DATA_BLOCK "Timer_ALARM_STOP_temp_DB"   // DB97
{ S7_Optimized_Access := 'TRUE' }
AUTHOR : Simatic
FAMILY : IEC
NAME : IEC_TMR
VERSION : 1.0
// stored: InstanceOfName IEC_TIMER
"IEC_TIMER"
BEGIN
END_DATA_BLOCK

DATA_BLOCK "Timer_PLAN_STOP_temp_DB"   // DB98
{ S7_Optimized_Access := 'TRUE' }
AUTHOR : Simatic
FAMILY : IEC
NAME : IEC_TMR
VERSION : 1.0
// stored: InstanceOfName IEC_TIMER
"IEC_TIMER"
BEGIN
END_DATA_BLOCK

DATA_BLOCK "Timer_IND_1_DB"   // DB100
{ S7_Optimized_Access := 'TRUE' }
AUTHOR : Simatic
FAMILY : IEC
NAME : IEC_TMR
VERSION : 1.0
// stored: InstanceOfName IEC_TIMER
"IEC_TIMER"
BEGIN
END_DATA_BLOCK

DATA_BLOCK "Timer_IND_2_DB"   // DB101
{ S7_Optimized_Access := 'TRUE' }
AUTHOR : Simatic
FAMILY : IEC
NAME : IEC_TMR
VERSION : 1.0
// stored: InstanceOfName IEC_TIMER
"IEC_TIMER"
BEGIN
END_DATA_BLOCK

DATA_BLOCK "TON_test_sound_DB"   // DB120
{ S7_Optimized_Access := 'TRUE' }
AUTHOR : Simatic
FAMILY : IEC
NAME : IEC_TMR
VERSION : 1.0
// stored: InstanceOfName IEC_TIMER
"IEC_TIMER"
BEGIN
END_DATA_BLOCK

DATA_BLOCK "TON_warning_1_DB"   // DB121
{ S7_Optimized_Access := 'TRUE' }
AUTHOR : Simatic
FAMILY : IEC
NAME : IEC_TMR
VERSION : 1.0
// stored: InstanceOfName IEC_TIMER
"IEC_TIMER"
BEGIN
END_DATA_BLOCK

DATA_BLOCK "TON_warning_2_DB"   // DB122
{ S7_Optimized_Access := 'TRUE' }
AUTHOR : Simatic
FAMILY : IEC
NAME : IEC_TMR
VERSION : 1.0
// stored: InstanceOfName IEC_TIMER
"IEC_TIMER"
BEGIN
END_DATA_BLOCK

DATA_BLOCK "Timer_RUN_temp_DB"   // DB124
{ S7_Optimized_Access := 'TRUE' }
AUTHOR : Simatic
FAMILY : IEC
NAME : IEC_LTMR
VERSION : 1.0
// stored: InstanceOfName IEC_LTIMER
"IEC_LTIMER"
BEGIN
END_DATA_BLOCK

// folder: (top level)

FUNCTION_BLOCK "PID_impulse"   // FB1, SCL
{ S7_Optimized_Access := 'FALSE' }
VERSION : 0.1
   VAR_INPUT
      DIR : Bool;   // Направление регулирования (1-позитивное,0-негативное)
      PV : Real;   // Величина параметра
      SP : Real;   // Величина уставки
      DB : Real;   // Зона нечувствительности
      KP : Real;   // ПИД Пропорциональный коэффициент
      TI : UDInt;   // ПИД Постоянная времени интегрирования (мс)
      TD : UDInt;   // ПИД Постоянная времени дифференцирования (мс)
      CYCLE : UDInt;   // Время цикла регулятора (мс)
      FMT : UDInt;   // Время хода исполнительного механизма (мс)
      DT_MIN : UDInt;   // Величина минимальной длительности импульса (мс)
      AUTO : Bool;   // Режим работы (0-ДИСТ, 1- АВТ)
      MORE : Bool;   // Дистанционное управление. Кнопка "Больше"
      LESS : Bool;   // Дистанционное управление. Кнопка "Меньше"
      Hold : Bool;   // (1-заморозка, 0-выполнение)
      GAP : DInt;   // Люфт
   END_VAR
   VAR_IN_OUT
      PLUS : Bool;   // Управление "Больше"
      MINUS : Bool;   // Управление "Меньше"
   END_VAR
   VAR
      BDP : Real;
      dD : Real;   // Приращение дифференциальной составляющей
      dD_max : Real;
      dI : Real;   // Приращение интегральной составляющей
      dP : Real;   // Приращение пропорциональной составляющей
      dP_1 : Real;
      dt10 : DInt;
      dt2_T : DInt;
      dt3 : DInt;
      dt3_T : DInt;
      dt4 : DInt;
      dt7 : DInt;
      dt8 : DInt;
      dt_imp_T : DInt;
      Err : Real;   // Ошибка рассогласования (t)
      Err_1 : Real;
      Err_1_T : Real;
      Ik : DInt;
      Int_reset : Bool;
      KPd : Real;
      L5 : Bool;
      L5_T : Bool;
      out : Bool;
      Pulse : Bool;   // Триггер импульса расчета
      Reset : Bool;
      TE : UDInt;   // Время цикла регулятора
      dP_T : Real;
      dI_T : Real;
      D_T : Real;
      A_N : Real := 8.0;
      A_Xf_1 : Real;
      A_Xf_2 : Real;
      D : Real;   // Приращение дифференциальной составляющей
      dD_1 : Real;
      dU : Real;   // Приращение управляющего воздействия
      dt1 : DInt;   // Длительность импульса
      dt6 : DInt;
      dt_imp : DInt;
      PLUS_T : Bool;
      MINUS_T : Bool;
      PAUSE : DInt;   // Время цикла регулятора
      L11 : Bool;
      L12 : Bool;
      Direct : Bool;   // Направление движения механизма (0-больше, 1-меньше)
   END_VAR
BEGIN
   (*Реальное время*)
   IF NOT #Reset THEN
       #TE := 0;
       #Reset := TRUE;
   ELSE
       #TE := #TE + "RT_INFO_DB".Cycle;
   END_IF;
   IF #TE >= #CYCLE AND #CYCLE <> 0 THEN
       #Pulse := TRUE;
   ELSE
       #Pulse := FALSE;
   END_IF;

   (*ПИД регулятор*)
   IF #Pulse THEN
       IF NOT #Hold THEN
           IF #AUTO THEN
               IF NOT #DIR THEN
                   #KPd := INT_TO_REAL(0) - #KP;
               ELSE
                   #KPd := #KP;
               END_IF;
               #Err := #SP - #PV;
               (*Зона нечувствительности*)
               IF ABS(#Err) < #DB / INT_TO_REAL(10) THEN
                   #Err_1 := INT_TO_REAL(0);
                   #Err_1_T := INT_TO_REAL(0);
               END_IF;
               IF ABS(#Err) > #DB / INT_TO_REAL(2) THEN
                   #Err_1 := #Err;
               END_IF;
               IF ABS(#Err) <= #DB / INT_TO_REAL(2) AND ABS(#Err) >= #DB / INT_TO_REAL(10) THEN
                   IF #Err_1_T = INT_TO_REAL(0) THEN
                       #Err_1 := INT_TO_REAL(0);
                       #Err_1_T := INT_TO_REAL(0);
                   ELSE
                       #Err_1 := #Err;
                   END_IF;
               END_IF;
               (*Д*)
               #dP := #KPd * (#Err_1 - #Err_1_T);
               (*Фильтрующий усилитель*)
               IF #TI > 0 THEN
                   #dI := #KPd * (UDINT_TO_REAL(#CYCLE) / UDINT_TO_REAL(#TI)) * ((#Err_1 + #Err_1_T) / INT_TO_REAL(2));
               ELSE
                   #dI := INT_TO_REAL(0);
               END_IF;
               (*ДД*)
               IF #TD > 0 THEN
                   (*Фильтр 1-го порядка (Апериодическое звено)*)
                   #A_Xf_1 := #A_Xf_1 + (#Err_1 - #A_Xf_1) * UDINT_TO_REAL(#CYCLE) / (UDINT_TO_REAL(#TD) / #A_N + UDINT_TO_REAL(#CYCLE));
                   (*Фильтр 2-го порядка (Апериодическое звено)*)
                   #A_Xf_2 := #A_Xf_2 + (#Err_1 - #A_Xf_1 - #A_Xf_2) * UDINT_TO_REAL(#CYCLE) / (UDINT_TO_REAL(#TD) / #A_N + UDINT_TO_REAL(#CYCLE));
                   #D := #KPd * #A_N * #A_Xf_2;
               ELSE
                   #A_Xf_1 := #Err_1;
                   #D := INT_TO_REAL(0);
               END_IF;
               #dD := #D - #D_T;
               (*Блокировка приращения пропорциональной составляющей*)
               #BDP := #KPd * #Err_1;
               IF #dP > INT_TO_REAL(0) AND #BDP < INT_TO_REAL(-100) THEN
                   #dP_1 := INT_TO_REAL(0);
               END_IF;
               IF #dP < INT_TO_REAL(0) AND #BDP > INT_TO_REAL(-100) THEN
                   #dP_1 := INT_TO_REAL(0);
               END_IF;
               IF ABS(#BDP) <= INT_TO_REAL(100) THEN
                   #dP_1 := #dP;
               END_IF;
               (*Ограничение приращений дифференциальной составляющей*)
               IF ABS(#dP_T + #dI_T) < INT_TO_REAL(100) THEN
                   #dD_max := INT_TO_REAL(100) - ABS(#dP_T + #dI_T);
               ELSE
                   #dD_max := INT_TO_REAL(0);
               END_IF;
               IF ABS(#dD) <= #dD_max THEN
                   #dD_1 := #dD;
               END_IF;
               IF #dD > #dD_max THEN
                   #dD_1 := #dD_max;
               END_IF;
               IF #dD < INT_TO_REAL(0) - #dD_max THEN
                   #dD_1 := INT_TO_REAL(0) - #dD_max;
               END_IF;
               (*Формирование ПИД закона*)
               #dU := #dP_1 + #dI + #dD_1;
               (*Ограничение амплитуды*)
               IF #dU < INT_TO_REAL(-100) THEN
                   #dU := INT_TO_REAL(-100);
               END_IF;
               IF #dU > INT_TO_REAL(100) THEN
                   #dU := INT_TO_REAL(100);
               END_IF;
               (*Расчет длительности импульса*)
               #dt1 := REAL_TO_DINT((UDINT_TO_REAL(#FMT) / INT_TO_REAL(100)) * #dU);
               (*Коррекция малых длительностей импульсов*)
               IF ABS(#dt1) < UDINT_TO_DINT(#DT_MIN) THEN
                   #dt3 := #dt1;
               ELSE
                   #dt3 := 0;
               END_IF;
               IF #dt2_T > UDINT_TO_DINT(#DT_MIN) AND ABS(#dt1) < UDINT_TO_DINT(#DT_MIN) THEN
                   #Int_reset := TRUE;
               ELSE
                   #Int_reset := FALSE;
               END_IF;
               #Ik := #Ik + #dt3;
               IF #Int_reset OR #L5_T THEN
                   #Ik := 0;
               END_IF;
               #dt4 := #dt1 + #Ik;
               IF ABS(#dt4) >= UDINT_TO_DINT(#DT_MIN) THEN
                   #L5 := TRUE;
               ELSE
                   #L5 := FALSE;
               END_IF;
               IF NOT #L5 THEN
                   #dt6 := #dt1;
               ELSE
                   #dt6 := #dt4;
               END_IF;
               (*Коррекция больших длительностей импульсов*)
               IF #dt_imp_T >= 0 THEN
                   #dt8 := UDINT_TO_DINT(#CYCLE) - #dt_imp_T;
               ELSE
                   #dt8 := - UDINT_TO_DINT(#CYCLE) - #dt_imp_T;
               END_IF;
               IF ABS(#dt8) > UDINT_TO_DINT(#CYCLE) THEN
                   #dt10 := #dt8;
               ELSE
                   #dt10 := 0;
               END_IF;
               #dt7 := #dt6 - #dt10;
               (*огр амп*)
               IF ABS(#dt7) <= UDINT_TO_DINT(#FMT) THEN
                   #dt_imp := #dt7;
               END_IF;
               IF #dt7 > UDINT_TO_DINT(#FMT) THEN
                   #dt_imp := UDINT_TO_DINT(#FMT);
               END_IF;
               IF #dt7 < - UDINT_TO_DINT(#FMT) THEN
                   #dt_imp := - UDINT_TO_DINT(#FMT);
               END_IF;
   (*Проверка ошибок*)
               ENO := TRUE;    //ENO := NOT P_ER;
           END_IF;
       ELSE
           #Err := INT_TO_REAL(0);
       END_IF;
       #Err_1_T := #Err_1;
       #dt2_T := ABS(#dt1);
       #dt3_T := #dt3;
       #dt_imp_T := #dt_imp;
       #L5_T := #L5;
       #dP_T := #dP;
       #dI_T := #dI;
       #D_T := #D;
       #TE := 0;
   END_IF;

   (* //компенсация люфта
   IF NOT #Direct AND #dt_imp < 0 THEN
       #dt_imp := #dt_imp - #GAP;
   END_IF;
   IF #Direct AND #dt_imp > 0 THEN
       #dt_imp := #dt_imp + #GAP;
   END_IF; *)

   (*Формирование ШИМ выхода*)
   IF #AUTO THEN
       IF UDINT_TO_DINT(#TE) >= ABS(#dt_imp) THEN
           #out := FALSE;
           #PLUS := false;
           #MINUS := false;
       ELSE
           #out := TRUE;
       END_IF;
       IF ABS(#dt_imp) >= UDINT_TO_DINT(#DT_MIN) THEN
           IF #dt_imp > 0 THEN
               IF #out THEN
                   #PLUS := true;
               ELSE
                   #PLUS := false;
               END_IF;
               #MINUS := false;
           ELSE
               IF #out THEN
                   #MINUS := true;
               ELSE
                   #MINUS := false;
               END_IF;
               #PLUS := false;
           END_IF;
   (*    ELSE
           #PLUS := false;
           #MINUS := false; *)
       END_IF;
   ELSE
       #PLUS := #MORE;
       #MINUS := #LESS;
   END_IF;
   (*Защита от частых коммутаций*)
   IF ((#PLUS_T AND NOT #PLUS) OR (#MINUS_T AND NOT #MINUS)) THEN
       #L11 := true;
   END_IF;
   IF #L11 THEN
       #PAUSE := UDINT_TO_DINT(#DT_MIN * INT_TO_UDINT(3));
       #L12 := true;
       #L11 := false;
   END_IF;
   IF #L12 THEN
       IF #PAUSE <= INT_TO_DINT(0) THEN
           #L12 := false;
           #PAUSE := INT_TO_DINT(0);
       ELSE
           #PAUSE := #PAUSE - UDINT_TO_DINT("RT_INFO_DB".Cycle); // / INT_TO_UDINT(10));
       END_IF;
   END_IF;
   IF #L12 AND #AUTO THEN
       #PLUS := false;
       #MINUS := false;
   END_IF;

   #PLUS_T := #PLUS;
   #MINUS_T := #MINUS;

   IF #PLUS THEN
       #Direct := FALSE;
   END_IF;
   IF #MINUS THEN
       #Direct := TRUE;
   END_IF;
END_FUNCTION_BLOCK

FUNCTION_BLOCK "PID_analog"   // FB2, SCL
{ S7_Optimized_Access := 'FALSE' }
VERSION : 0.1
   VAR_INPUT
      AUTO : Bool;   // Mode (0-manual, 1-automatic)
      DIR : Bool;   // Direction (1-positive,0-negative)
      PV : Real;   // Process variable
      SP : Real;   // Setpoint
      DB : Real;   // Deadband
      KP : Real;   // Proportional constant
      TI : UDInt;   // Integral time constant (ms)
      TD : UDInt;   // Derivative time constant (ms)
      CYCLE : UDInt;   // Cycle time (ms)
      OUT_MIN : Real;   // Output min limit (automatic mode)
      OUT_MAX : Real := 100.0;   // Output max limit (automatic mode)
      OUT_MAN : Real;   // Output (manual mode)
      Hold : Bool;   // (1-заморозка, 0-выполнение)
   END_VAR
   VAR_IN_OUT
      OUT : Real;   // Output control
   END_VAR
   VAR
      Err : Real;   // Ошибка рассогласования (t)
      Err_T : Real;   // Предыдущее значение ошибки рассогласования (t-1)
      Out_T : Real;   // Предыдущее значение выхода (t-1)
      Er : Real;   // Ошибка рассогласования (t)
      Er_T : Real;   // Предыдущее значение ошибки рассогласования (t-1)
      Integral : Real;   // Интегральная составляющая (t)
      Integral_T : Real;   // Интегральная составляющая (t-1)
      Integral_D : Real;   // Интегральное изменение
      Pulse : Bool;   // Триггер импульса расчета
      TE : UDInt;
      Reset : Bool;
      KPd : Real;
      A_N : Real := 8.0;
      A_Xf_1 : Real;
      A_Xf_2 : Real;
      Diff : Real;
   END_VAR
BEGIN
   (*Реальное время*)
   IF NOT #Reset THEN
       #TE := 0;
       #Reset := TRUE;
   ELSE
       #TE := #TE + "RT_INFO_DB".Cycle;
   END_IF;
   IF #TE >= #CYCLE AND #CYCLE <> 0 THEN
       #Pulse := TRUE;
   ELSE
       #Pulse := FALSE;
   END_IF;

   (*ПИД регулятор*)
   IF #Pulse THEN
       #Err := #SP - #PV;
       #Er := #Err;
       IF NOT #Hold THEN
           IF NOT #DIR THEN
               #KPd := INT_TO_REAL(0) - #KP;
           ELSE
               #KPd := #KP;
           END_IF;
           IF #AUTO THEN
               IF ABS(#Er) < #DB / INT_TO_REAL(10) THEN
                   #Err := INT_TO_REAL(0);
                   #Err_T := INT_TO_REAL(0);
               END_IF;
               IF ABS(#Er) > #DB / INT_TO_REAL(2) THEN
                   #Err := #Er;
               END_IF;
               IF ABS(#Er) <= #DB / INT_TO_REAL(2) AND ABS(#Er) >= #DB / INT_TO_REAL(10) THEN
                   IF #Err_T = INT_TO_REAL(0) THEN
                       #Err := INT_TO_REAL(0);
                       #Err_T := INT_TO_REAL(0);
                   ELSE
                       #Err := #Er;
                   END_IF;
               END_IF;
               IF #TI <= 0 THEN
                   #Integral_T := INT_TO_REAL(0);
                   #Integral_D := INT_TO_REAL(0);
                   #Integral := INT_TO_REAL(0);
               ELSE
                   #Integral_D := #KPd * ((#Err * UDINT_TO_REAL(#TE)) / UDINT_TO_REAL(#TI));
                   #Integral := #Integral_T + #Integral_D;
               END_IF;
               IF #TD > 0 THEN
                   (*Фильтр 1-го порядка (Апериодическое звено)*)
                   #A_Xf_1 := #A_Xf_1 + (#Err - #A_Xf_1) * UDINT_TO_REAL(#TE) / (UDINT_TO_REAL(#TD) / #A_N + UDINT_TO_REAL(#TE));
                   (*Фильтр 2-го порядка (Апериодическое звено)*)
                   #A_Xf_2 := #A_Xf_2 + (#Err - #A_Xf_1 - #A_Xf_2) * UDINT_TO_REAL(#TE) / (UDINT_TO_REAL(#TD) / #A_N + UDINT_TO_REAL(#TE));
                   #Diff := #KPd * #A_N * #A_Xf_2;
               ELSE
                   #A_Xf_1 := #Err;
                   #Diff := INT_TO_REAL(0);
               END_IF;
               #OUT := #KPd * #Err + #Integral + #Diff;
               IF #OUT < #OUT_MIN THEN
                   IF #Integral_D < INT_TO_REAL(0) THEN
                       #Integral_D := INT_TO_REAL(0);
                   END_IF;
               END_IF;
               IF #OUT > #OUT_MAX THEN
                   IF #Integral_D > INT_TO_REAL(0) THEN
                       #Integral_D := INT_TO_REAL(0);
                   END_IF;
               END_IF;
               #Integral := #Integral_T + #Integral_D;
               #OUT := #KPd * #Err + #Integral + #Diff;
               IF #OUT < #OUT_MIN THEN
                   #OUT := #OUT_MIN;
               END_IF;
               IF #OUT > #OUT_MAX THEN
                   #OUT := #OUT_MAX;
               END_IF;
           ELSE
               #OUT := #OUT_MAN;
               IF #OUT < #OUT_MIN THEN
                   #OUT := #OUT_MIN;
               END_IF;
               IF #OUT > #OUT_MAX THEN
                   #OUT := #OUT_MAX;
               END_IF;
               #Integral := #OUT - #KPd * #Err;
               #A_Xf_1 := INT_TO_REAL(0);
               #A_Xf_2 := INT_TO_REAL(0);
           END_IF;
           (*Проверка ошибок*)
           ENO := TRUE;    //ENO := NOT P_ER;
       ELSE
           #Err := INT_TO_REAL(0);
           #Err_T := INT_TO_REAL(0);
           #OUT := #OUT_MIN;
           #Integral := INT_TO_REAL(0);
       END_IF;
       #Err_T := #Err;
       #Er_T := #Er;
       #Out_T := #OUT;
       #Integral_T := #Integral;
       #TE := 0;
   END_IF;
END_FUNCTION_BLOCK

FUNCTION_BLOCK "TIME_converter"   // FB3, SCL
{ S7_Optimized_Access := 'TRUE' }
VERSION : 0.1
   VAR_INPUT
      IN : Time;   // входная переменная тип Time
   END_VAR
   VAR_OUTPUT
      Hour : Int;   // Часы
      Minute : Int;   // Минуты
      Second : Int;   // Секунды
   END_VAR
   VAR_TEMP
      in_dint_ms : DInt;
      in_dint_s : DInt;
      in_dint_m : DInt;
      in_dint_h : DInt;
   END_VAR
BEGIN
   #in_dint_ms := T_CONV(#IN);
   #in_dint_s := #in_dint_ms / 1000;
   #in_dint_m := #in_dint_s / 60;
   #in_dint_h := #in_dint_m / 60;

   #Second := DINT_TO_INT((#in_dint_s) MOD (60));
   #Minute := DINT_TO_INT((#in_dint_m) MOD (60));
   #Hour := DINT_TO_INT(#in_dint_h);
END_FUNCTION_BLOCK

FUNCTION_BLOCK "LTIME_converter"   // FB4, SCL
{ S7_Optimized_Access := 'TRUE' }
VERSION : 0.1
   VAR_INPUT
      IN : LTime;   // входная переменная тип LTime
   END_VAR
   VAR_OUTPUT
      Day : DInt;   // Дни
      Hour : Int;   // Часы
      Minute : Int;   // Минуты
      Second : Int;   // Секунды
      mSecond : Int;   // Миллисекунды
      uSecond : Int;   // Микросекунды
      nSecond : Int;   // Наносекунды
   END_VAR
   VAR_TEMP
      temp_ns : LInt;
      temp_us : LInt;
      temp_ms : LInt;
      temp_s : LInt;
      temp_m : LInt;
      temp_h : LInt;
      temp_d : LInt;
   END_VAR
BEGIN
   #temp_ns := T_CONV(#IN);
   #temp_us := #temp_ns / 1000;
   #temp_ms := #temp_us / 1000;
   #temp_s := #temp_ms / 1000;
   #temp_m := #temp_s / 60;
   #temp_h := #temp_m / 60;
   #temp_d := #temp_h / 24;

   #nSecond := LINT_TO_INT((#temp_ns) MOD (1000));
   #uSecond := LINT_TO_INT((#temp_us) MOD (1000));
   #mSecond := LINT_TO_INT((#temp_ms) MOD (1000));
   #Second := LINT_TO_INT((#temp_s) MOD (60));
   #Minute := LINT_TO_INT((#temp_m) MOD (60));
   #Hour := LINT_TO_INT((#temp_h) MOD (24));
   #Day := LINT_TO_DINT(#temp_d);
END_FUNCTION_BLOCK

FUNCTION "Read_inputs" : Void   // FC1, SCL
{ S7_Optimized_Access := 'TRUE' }
VERSION : 0.1
BEGIN
   (*ЧТЕНИЕ ВХОДОВ*)
   (*Чтение аналоговых входов*)
   (*Температура сетевой воды перед котлом*)
   IF "Sensors".T_water_before_boiler.Enable THEN
       "Read_sensor_4_20"(N_module := "Sensors".T_water_before_boiler.N_module,
                          N_chanel := "Sensors".T_water_before_boiler.N_chanel,
                          Low_limit_phisical_current := "Sensors".T_water_before_boiler.Low_limit_phisical_current,
                          High_limit_phisical_current := "Sensors".T_water_before_boiler.High_limit_phisical_current,
                          Low_limit_ADC_current := "Sensors".T_water_before_boiler.Low_limit_ADC_current,
                          High_limit_ADC_current := "Sensors".T_water_before_boiler.High_limit_ADC_current,
                          Current_ADC => "Sensors".T_water_before_boiler.Current_ADC,
                          Value => "Sensors".T_water_before_boiler.Value,
                          Alarm_sensor => "Sensors".T_water_before_boiler.Alarm_sensor,
                          Current => "Sensors".T_water_before_boiler.Current);
       //применение изменений значений точек для пересчета сигнала
       IF "Sensors".T_water_before_boiler.Apply THEN
           "Sensors".T_water_before_boiler.Low_limit_phisical_current := "Sensors".T_water_before_boiler.Low_limit_phisical_new;
           "Sensors".T_water_before_boiler.High_limit_phisical_current := "Sensors".T_water_before_boiler.High_limit_phisical_new;
           "Sensors".T_water_before_boiler.Low_limit_ADC_current := "Sensors".T_water_before_boiler.Low_limit_ADC_new;
           "Sensors".T_water_before_boiler.High_limit_ADC_current := "Sensors".T_water_before_boiler.High_limit_ADC_new;
           "Sensors".T_water_before_boiler.Apply := false;
       END_IF;
   ELSE
       "Sensors".T_water_before_boiler.Apply := false;
   END_IF;

   (*Давление сетевой воды перед котлом*)
   IF "Sensors".P_water_before_boiler.Enable THEN
       "Read_sensor_4_20"(N_module := "Sensors".P_water_before_boiler.N_module,
                          N_chanel := "Sensors".P_water_before_boiler.N_chanel,
                          Low_limit_phisical_current := "Sensors".P_water_before_boiler.Low_limit_phisical_current,
                          High_limit_phisical_current := "Sensors".P_water_before_boiler.High_limit_phisical_current,
                          Low_limit_ADC_current := "Sensors".P_water_before_boiler.Low_limit_ADC_current,
                          High_limit_ADC_current := "Sensors".P_water_before_boiler.High_limit_ADC_current,
                          Current_ADC => "Sensors".P_water_before_boiler.Current_ADC,
                          Value => "Sensors".P_water_before_boiler.Value,
                          Alarm_sensor => "Sensors".P_water_before_boiler.Alarm_sensor,
                          Current => "Sensors".P_water_before_boiler.Current);
       //применение изменений значений точек для пересчета сигнала
       IF "Sensors".P_water_before_boiler.Apply THEN
           "Sensors".P_water_before_boiler.Low_limit_phisical_current := "Sensors".P_water_before_boiler.Low_limit_phisical_new;
           "Sensors".P_water_before_boiler.High_limit_phisical_current := "Sensors".P_water_before_boiler.High_limit_phisical_new;
           "Sensors".P_water_before_boiler.Low_limit_ADC_current := "Sensors".P_water_before_boiler.Low_limit_ADC_new;
           "Sensors".P_water_before_boiler.High_limit_ADC_current := "Sensors".P_water_before_boiler.High_limit_ADC_new;
           "Sensors".P_water_before_boiler.Apply := false;
       END_IF;
   ELSE
       "Sensors".P_water_before_boiler.Apply := false;
   END_IF;

   (*Перепад давления сетевой воды через котел (кПа)*)
   IF "Sensors".dP_water_boiler.Enable THEN
       "Read_sensor_4_20"(N_module := "Sensors".dP_water_boiler.N_module,
                          N_chanel := "Sensors".dP_water_boiler.N_chanel,
                          Low_limit_phisical_current := "Sensors".dP_water_boiler.Low_limit_phisical_current,
                          High_limit_phisical_current := "Sensors".dP_water_boiler.High_limit_phisical_current,
                          Low_limit_ADC_current := "Sensors".dP_water_boiler.Low_limit_ADC_current,
                          High_limit_ADC_current := "Sensors".dP_water_boiler.High_limit_ADC_current,
                          Current_ADC => "Sensors".dP_water_boiler.Current_ADC,
                          Value => "Sensors".dP_water_boiler.Value,
                          Alarm_sensor => "Sensors".dP_water_boiler.Alarm_sensor,
                          Current => "Sensors".dP_water_boiler.Current);
       //применение изменений значений точек для пересчета сигнала
       IF "Sensors".dP_water_boiler.Apply THEN
           "Sensors".dP_water_boiler.Low_limit_phisical_current := "Sensors".dP_water_boiler.Low_limit_phisical_new;
           "Sensors".dP_water_boiler.High_limit_phisical_current := "Sensors".dP_water_boiler.High_limit_phisical_new;
           "Sensors".dP_water_boiler.Low_limit_ADC_current := "Sensors".dP_water_boiler.Low_limit_ADC_new;
           "Sensors".dP_water_boiler.High_limit_ADC_current := "Sensors".dP_water_boiler.High_limit_ADC_new;
           "Sensors".dP_water_boiler.Apply := false;
       END_IF;
   ELSE
       "Sensors".dP_water_boiler.Apply := false;
   END_IF;

   (*Температура сетевой воды после котла*)
   IF "Sensors".T_water_after_boiler.Enable THEN
       "Read_sensor_4_20"(N_module := "Sensors".T_water_after_boiler.N_module,
                          N_chanel := "Sensors".T_water_after_boiler.N_chanel,
                          Low_limit_phisical_current := "Sensors".T_water_after_boiler.Low_limit_phisical_current,
                          High_limit_phisical_current := "Sensors".T_water_after_boiler.High_limit_phisical_current,
                          Low_limit_ADC_current := "Sensors".T_water_after_boiler.Low_limit_ADC_current,
                          High_limit_ADC_current := "Sensors".T_water_after_boiler.High_limit_ADC_current,
                          Current_ADC => "Sensors".T_water_after_boiler.Current_ADC,
                          Value => "Sensors".T_water_after_boiler.Value,
                          Alarm_sensor => "Sensors".T_water_after_boiler.Alarm_sensor,
                          Current => "Sensors".T_water_after_boiler.Current);
       //применение изменений значений точек для пересчета сигнала
       IF "Sensors".T_water_after_boiler.Apply THEN
           "Sensors".T_water_after_boiler.Low_limit_phisical_current := "Sensors".T_water_after_boiler.Low_limit_phisical_new;
           "Sensors".T_water_after_boiler.High_limit_phisical_current := "Sensors".T_water_after_boiler.High_limit_phisical_new;
           "Sensors".T_water_after_boiler.Low_limit_ADC_current := "Sensors".T_water_after_boiler.Low_limit_ADC_new;
           "Sensors".T_water_after_boiler.High_limit_ADC_current := "Sensors".T_water_after_boiler.High_limit_ADC_new;
           "Sensors".T_water_after_boiler.Apply := false;
       END_IF;
   ELSE
       "Sensors".T_water_after_boiler.Apply := false;
   END_IF;

   (*Давление сетевой воды после котла*)
   IF "Sensors".P_water_after_boiler.Enable THEN
       "Read_sensor_4_20"(N_module := "Sensors".P_water_after_boiler.N_module,
                          N_chanel := "Sensors".P_water_after_boiler.N_chanel,
                          Low_limit_phisical_current := "Sensors".P_water_after_boiler.Low_limit_phisical_current,
                          High_limit_phisical_current := "Sensors".P_water_after_boiler.High_limit_phisical_current,
                          Low_limit_ADC_current := "Sensors".P_water_after_boiler.Low_limit_ADC_current,
                          High_limit_ADC_current := "Sensors".P_water_after_boiler.High_limit_ADC_current,
                          Current_ADC => "Sensors".P_water_after_boiler.Current_ADC,
                          Value => "Sensors".P_water_after_boiler.Value,
                          Alarm_sensor => "Sensors".P_water_after_boiler.Alarm_sensor,
                          Current => "Sensors".P_water_after_boiler.Current);
       //применение изменений значений точек для пересчета сигнала
       IF "Sensors".P_water_after_boiler.Apply THEN
           "Sensors".P_water_after_boiler.Low_limit_phisical_current := "Sensors".P_water_after_boiler.Low_limit_phisical_new;
           "Sensors".P_water_after_boiler.High_limit_phisical_current := "Sensors".P_water_after_boiler.High_limit_phisical_new;
           "Sensors".P_water_after_boiler.Low_limit_ADC_current := "Sensors".P_water_after_boiler.Low_limit_ADC_new;
           "Sensors".P_water_after_boiler.High_limit_ADC_current := "Sensors".P_water_after_boiler.High_limit_ADC_new;
           "Sensors".P_water_after_boiler.Apply := false;
       END_IF;
   ELSE
       "Sensors".P_water_after_boiler.Apply := false;
   END_IF;

   (*Перепад давления сетевой воды через котел (кПа)*)
   IF "Sensors".dP_water_boiler_1.Enable THEN
       "Read_sensor_4_20"(N_module := "Sensors".dP_water_boiler_1.N_module,
                          N_chanel := "Sensors".dP_water_boiler_1.N_chanel,
                          Low_limit_phisical_current := "Sensors".dP_water_boiler_1.Low_limit_phisical_current,
                          High_limit_phisical_current := "Sensors".dP_water_boiler_1.High_limit_phisical_current,
                          Low_limit_ADC_current := "Sensors".dP_water_boiler_1.Low_limit_ADC_current,
                          High_limit_ADC_current := "Sensors".dP_water_boiler_1.High_limit_ADC_current,
                          Current_ADC => "Sensors".dP_water_boiler_1.Current_ADC,
                          Value => "Sensors".dP_water_boiler_1.Value,
                          Alarm_sensor => "Sensors".dP_water_boiler_1.Alarm_sensor,
                          Current => "Sensors".dP_water_boiler_1.Current);
       //применение изменений значений точек для пересчета сигнала
       IF "Sensors".dP_water_boiler_1.Apply THEN
           "Sensors".dP_water_boiler_1.Low_limit_phisical_current := "Sensors".dP_water_boiler_1.Low_limit_phisical_new;
           "Sensors".dP_water_boiler_1.High_limit_phisical_current := "Sensors".dP_water_boiler_1.High_limit_phisical_new;
           "Sensors".dP_water_boiler_1.Low_limit_ADC_current := "Sensors".dP_water_boiler_1.Low_limit_ADC_new;
           "Sensors".dP_water_boiler_1.High_limit_ADC_current := "Sensors".dP_water_boiler_1.High_limit_ADC_new;
           "Sensors".dP_water_boiler_1.Apply := false;
       END_IF;
   ELSE
       "Sensors".dP_water_boiler_1.Apply := false;
   END_IF;

   (*Давление сетевой воды перед котлом*)
   IF "Sensors".P_water_before_boiler_1.Enable THEN
       "Read_sensor_4_20"(N_module := "Sensors".P_water_before_boiler_1.N_module,
                          N_chanel := "Sensors".P_water_before_boiler_1.N_chanel,
                          Low_limit_phisical_current := "Sensors".P_water_before_boiler_1.Low_limit_phisical_current,
                          High_limit_phisical_current := "Sensors".P_water_before_boiler_1.High_limit_phisical_current,
                          Low_limit_ADC_current := "Sensors".P_water_before_boiler_1.Low_limit_ADC_current,
                          High_limit_ADC_current := "Sensors".P_water_before_boiler_1.High_limit_ADC_current,
                          Current_ADC => "Sensors".P_water_before_boiler_1.Current_ADC,
                          Value => "Sensors".P_water_before_boiler_1.Value,
                          Alarm_sensor => "Sensors".P_water_before_boiler_1.Alarm_sensor,
                          Current => "Sensors".P_water_before_boiler_1.Current);
       //применение изменений значений точек для пересчета сигнала
       IF "Sensors".P_water_before_boiler_1.Apply THEN
           "Sensors".P_water_before_boiler_1.Low_limit_phisical_current := "Sensors".P_water_before_boiler_1.Low_limit_phisical_new;
           "Sensors".P_water_before_boiler_1.High_limit_phisical_current := "Sensors".P_water_before_boiler_1.High_limit_phisical_new;
           "Sensors".P_water_before_boiler_1.Low_limit_ADC_current := "Sensors".P_water_before_boiler_1.Low_limit_ADC_new;
           "Sensors".P_water_before_boiler_1.High_limit_ADC_current := "Sensors".P_water_before_boiler_1.High_limit_ADC_new;
           "Sensors".P_water_before_boiler_1.Apply := false;
       END_IF;
   ELSE
       "Sensors".P_water_before_boiler_1.Apply := false;
   END_IF;

   (*dP газа на котел*)
   IF "Sensors".dP_gas_boiler.Enable THEN
       "Read_sensor_4_20"(N_module := "Sensors".dP_gas_boiler.N_module,
                          N_chanel := "Sensors".dP_gas_boiler.N_chanel,
                          Low_limit_phisical_current := "Sensors".dP_gas_boiler.Low_limit_phisical_current,
                          High_limit_phisical_current := "Sensors".dP_gas_boiler.High_limit_phisical_current,
                          Low_limit_ADC_current := "Sensors".dP_gas_boiler.Low_limit_ADC_current,
                          High_limit_ADC_current := "Sensors".dP_gas_boiler.High_limit_ADC_current,
                          Current_ADC => "Sensors".dP_gas_boiler.Current_ADC,
                          Value => "Sensors".dP_gas_boiler.Value,
                          Alarm_sensor => "Sensors".dP_gas_boiler.Alarm_sensor,
                          Current => "Sensors".dP_gas_boiler.Current);
       //применение изменений значений точек для пересчета сигнала
       IF "Sensors".dP_gas_boiler.Apply THEN
           "Sensors".dP_gas_boiler.Low_limit_phisical_current := "Sensors".dP_gas_boiler.Low_limit_phisical_new;
           "Sensors".dP_gas_boiler.High_limit_phisical_current := "Sensors".dP_gas_boiler.High_limit_phisical_new;
           "Sensors".dP_gas_boiler.Low_limit_ADC_current := "Sensors".dP_gas_boiler.Low_limit_ADC_new;
           "Sensors".dP_gas_boiler.High_limit_ADC_current := "Sensors".dP_gas_boiler.High_limit_ADC_new;
           "Sensors".dP_gas_boiler.Apply := false;
       END_IF;
   ELSE
       "Sensors".dP_gas_boiler.Apply := false;
   END_IF;

   (*Разрежение в топке котла*)
   IF "Sensors".dP_furnace_boiler.Enable THEN
       "Read_sensor_4_20"(N_module := "Sensors".dP_furnace_boiler.N_module,
                          N_chanel := "Sensors".dP_furnace_boiler.N_chanel,
                          Low_limit_phisical_current := "Sensors".dP_furnace_boiler.Low_limit_phisical_current,
                          High_limit_phisical_current := "Sensors".dP_furnace_boiler.High_limit_phisical_current,
                          Low_limit_ADC_current := "Sensors".dP_furnace_boiler.Low_limit_ADC_current,
                          High_limit_ADC_current := "Sensors".dP_furnace_boiler.High_limit_ADC_current,
                          Current_ADC => "Sensors".dP_furnace_boiler.Current_ADC,
                          Value => "Sensors".dP_furnace_boiler.Value,
                          Alarm_sensor => "Sensors".dP_furnace_boiler.Alarm_sensor,
                          Current => "Sensors".dP_furnace_boiler.Current);
       //применение изменений значений точек для пересчета сигнала
       IF "Sensors".dP_furnace_boiler.Apply THEN
           "Sensors".dP_furnace_boiler.Low_limit_phisical_current := "Sensors".dP_furnace_boiler.Low_limit_phisical_new;
           "Sensors".dP_furnace_boiler.High_limit_phisical_current := "Sensors".dP_furnace_boiler.High_limit_phisical_new;
           "Sensors".dP_furnace_boiler.Low_limit_ADC_current := "Sensors".dP_furnace_boiler.Low_limit_ADC_new;
           "Sensors".dP_furnace_boiler.High_limit_ADC_current := "Sensors".dP_furnace_boiler.High_limit_ADC_new;
           "Sensors".dP_furnace_boiler.Apply := false;
       END_IF;
   ELSE
       "Sensors".dP_furnace_boiler.Apply := false;
   END_IF;

   (*Давление газа между ПЗК-1 и ПЗК-2*)
   IF "Sensors".P_gas_before_PZK1_and_PZK2.Enable THEN
       "Read_sensor_4_20"(N_module := "Sensors".P_gas_before_PZK1_and_PZK2.N_module,
                          N_chanel := "Sensors".P_gas_before_PZK1_and_PZK2.N_chanel,
                          Low_limit_phisical_current := "Sensors".P_gas_before_PZK1_and_PZK2.Low_limit_phisical_current,
                          High_limit_phisical_current := "Sensors".P_gas_before_PZK1_and_PZK2.High_limit_phisical_current,
                          Low_limit_ADC_current := "Sensors".P_gas_before_PZK1_and_PZK2.Low_limit_ADC_current,
                          High_limit_ADC_current := "Sensors".P_gas_before_PZK1_and_PZK2.High_limit_ADC_current,
                          Current_ADC => "Sensors".P_gas_before_PZK1_and_PZK2.Current_ADC,
                          Value => "Sensors".P_gas_before_PZK1_and_PZK2.Value,
                          Alarm_sensor => "Sensors".P_gas_before_PZK1_and_PZK2.Alarm_sensor,
                          Current => "Sensors".P_gas_before_PZK1_and_PZK2.Current);
       //применение изменений значений точек для пересчета сигнала
       IF "Sensors".P_gas_before_PZK1_and_PZK2.Apply THEN
           "Sensors".P_gas_before_PZK1_and_PZK2.Low_limit_phisical_current := "Sensors".P_gas_before_PZK1_and_PZK2.Low_limit_phisical_new;
           "Sensors".P_gas_before_PZK1_and_PZK2.High_limit_phisical_current := "Sensors".P_gas_before_PZK1_and_PZK2.High_limit_phisical_new;
           "Sensors".P_gas_before_PZK1_and_PZK2.Low_limit_ADC_current := "Sensors".P_gas_before_PZK1_and_PZK2.Low_limit_ADC_new;
           "Sensors".P_gas_before_PZK1_and_PZK2.High_limit_ADC_current := "Sensors".P_gas_before_PZK1_and_PZK2.High_limit_ADC_new;
           "Sensors".P_gas_before_PZK1_and_PZK2.Apply := false;
       END_IF;
   ELSE
       "Sensors".P_gas_before_PZK1_and_PZK2.Apply := false;
   END_IF;

   (*Давление газа перед горелкой*)
   IF "Sensors".P_gas_before_burner.Enable THEN
       "Read_sensor_4_20"(N_module := "Sensors".P_gas_before_burner.N_module,
                          N_chanel := "Sensors".P_gas_before_burner.N_chanel,
                          Low_limit_phisical_current := "Sensors".P_gas_before_burner.Low_limit_phisical_current,
                          High_limit_phisical_current := "Sensors".P_gas_before_burner.High_limit_phisical_current,
                          Low_limit_ADC_current := "Sensors".P_gas_before_burner.Low_limit_ADC_current,
                          High_limit_ADC_current := "Sensors".P_gas_before_burner.High_limit_ADC_current,
                          Current_ADC => "Sensors".P_gas_before_burner.Current_ADC,
                          Value => "Sensors".P_gas_before_burner.Value,
                          Alarm_sensor => "Sensors".P_gas_before_burner.Alarm_sensor,
                          Current => "Sensors".P_gas_before_burner.Current);
       //применение изменений значений точек для пересчета сигнала
       IF "Sensors".P_gas_before_burner.Apply THEN
           "Sensors".P_gas_before_burner.Low_limit_phisical_current := "Sensors".P_gas_before_burner.Low_limit_phisical_new;
           "Sensors".P_gas_before_burner.High_limit_phisical_current := "Sensors".P_gas_before_burner.High_limit_phisical_new;
           "Sensors".P_gas_before_burner.Low_limit_ADC_current := "Sensors".P_gas_before_burner.Low_limit_ADC_new;
           "Sensors".P_gas_before_burner.High_limit_ADC_current := "Sensors".P_gas_before_burner.High_limit_ADC_new;
           "Sensors".P_gas_before_burner.Apply := false;
       END_IF;
   ELSE
       "Sensors".P_gas_before_burner.Apply := false;
   END_IF;

   (*Давление воздуха к горелке*)
   IF "Sensors".P_air_burner.Enable THEN
       "Read_sensor_4_20"(N_module := "Sensors".P_air_burner.N_module,
                          N_chanel := "Sensors".P_air_burner.N_chanel,
                          Low_limit_phisical_current := "Sensors".P_air_burner.Low_limit_phisical_current,
                          High_limit_phisical_current := "Sensors".P_air_burner.High_limit_phisical_current,
                          Low_limit_ADC_current := "Sensors".P_air_burner.Low_limit_ADC_current,
                          High_limit_ADC_current := "Sensors".P_air_burner.High_limit_ADC_current,
                          Current_ADC => "Sensors".P_air_burner.Current_ADC,
                          Value => "Sensors".P_air_burner.Value,
                          Alarm_sensor => "Sensors".P_air_burner.Alarm_sensor,
                          Current => "Sensors".P_air_burner.Current);
       //применение изменений значений точек для пересчета сигнала
       IF "Sensors".P_air_burner.Apply THEN
           "Sensors".P_air_burner.Low_limit_phisical_current := "Sensors".P_air_burner.Low_limit_phisical_new;
           "Sensors".P_air_burner.High_limit_phisical_current := "Sensors".P_air_burner.High_limit_phisical_new;
           "Sensors".P_air_burner.Low_limit_ADC_current := "Sensors".P_air_burner.Low_limit_ADC_new;
           "Sensors".P_air_burner.High_limit_ADC_current := "Sensors".P_air_burner.High_limit_ADC_new;
           "Sensors".P_air_burner.Apply := false;
       END_IF;
   ELSE
       "Sensors".P_air_burner.Apply := false;
   END_IF;

   (*Температура уходящих газов*)
   IF "Sensors".T_exhaust_gas.Enable THEN
       "Read_sensor_4_20"(N_module := "Sensors".T_exhaust_gas.N_module,
                          N_chanel := "Sensors".T_exhaust_gas.N_chanel,
                          Low_limit_phisical_current := "Sensors".T_exhaust_gas.Low_limit_phisical_current,
                          High_limit_phisical_current := "Sensors".T_exhaust_gas.High_limit_phisical_current,
                          Low_limit_ADC_current := "Sensors".T_exhaust_gas.Low_limit_ADC_current,
                          High_limit_ADC_current := "Sensors".T_exhaust_gas.High_limit_ADC_current,
                          Current_ADC => "Sensors".T_exhaust_gas.Current_ADC,
                          Value => "Sensors".T_exhaust_gas.Value,
                          Alarm_sensor => "Sensors".T_exhaust_gas.Alarm_sensor,
                          Current => "Sensors".T_exhaust_gas.Current);
       //применение изменений значений точек для пересчета сигнала
       IF "Sensors".T_exhaust_gas.Apply THEN
           "Sensors".T_exhaust_gas.Low_limit_phisical_current := "Sensors".T_exhaust_gas.Low_limit_phisical_new;
           "Sensors".T_exhaust_gas.High_limit_phisical_current := "Sensors".T_exhaust_gas.High_limit_phisical_new;
           "Sensors".T_exhaust_gas.Low_limit_ADC_current := "Sensors".T_exhaust_gas.Low_limit_ADC_new;
           "Sensors".T_exhaust_gas.High_limit_ADC_current := "Sensors".T_exhaust_gas.High_limit_ADC_new;
           "Sensors".T_exhaust_gas.Apply := false;
       END_IF;
   ELSE
       "Sensors".T_exhaust_gas.Apply := false;
   END_IF;

   (*Положение рег. заслонки газа перед котлом*)
   IF "Sensors".ZRG_position.Enable THEN
       "Read_sensor_4_20"(N_module := "Sensors".ZRG_position.N_module,
                          N_chanel := "Sensors".ZRG_position.N_chanel,
                          Low_limit_phisical_current := "Sensors".ZRG_position.Low_limit_phisical_current,
                          High_limit_phisical_current := "Sensors".ZRG_position.High_limit_phisical_current,
                          Low_limit_ADC_current := "Sensors".ZRG_position.Low_limit_ADC_current,
                          High_limit_ADC_current := "Sensors".ZRG_position.High_limit_ADC_current,
                          Current_ADC => "Sensors".ZRG_position.Current_ADC,
                          Value => "Sensors".ZRG_position.Value,
                          Alarm_sensor => "Sensors".ZRG_position.Alarm_sensor,
                          Current => "Sensors".ZRG_position.Current);
       //применение изменений значений точек для пересчета сигнала
       IF "Sensors".ZRG_position.Apply THEN
           "Sensors".ZRG_position.Low_limit_phisical_current := "Sensors".ZRG_position.Low_limit_phisical_new;
           "Sensors".ZRG_position.High_limit_phisical_current := "Sensors".ZRG_position.High_limit_phisical_new;
           "Sensors".ZRG_position.Low_limit_ADC_current := "Sensors".ZRG_position.Low_limit_ADC_new;
           "Sensors".ZRG_position.High_limit_ADC_current := "Sensors".ZRG_position.High_limit_ADC_new;
           "Sensors".ZRG_position.Apply := false;
       END_IF;
   ELSE
       "Sensors".ZRG_position.Apply := false;
   END_IF;

   (*Положение направл. аппарата вентилятора*)
   IF "Sensors".NAV_position.Enable THEN
       "Read_sensor_4_20"(N_module := "Sensors".NAV_position.N_module,
                          N_chanel := "Sensors".NAV_position.N_chanel,
                          Low_limit_phisical_current := "Sensors".NAV_position.Low_limit_phisical_current,
                          High_limit_phisical_current := "Sensors".NAV_position.High_limit_phisical_current,
                          Low_limit_ADC_current := "Sensors".NAV_position.Low_limit_ADC_current,
                          High_limit_ADC_current := "Sensors".NAV_position.High_limit_ADC_current,
                          Current_ADC => "Sensors".NAV_position.Current_ADC,
                          Value => "Sensors".NAV_position.Value,
                          Alarm_sensor => "Sensors".NAV_position.Alarm_sensor,
                          Current => "Sensors".NAV_position.Current);
       //применение изменений значений точек для пересчета сигнала
       IF "Sensors".NAV_position.Apply THEN
           "Sensors".NAV_position.Low_limit_phisical_current := "Sensors".NAV_position.Low_limit_phisical_new;
           "Sensors".NAV_position.High_limit_phisical_current := "Sensors".NAV_position.High_limit_phisical_new;
           "Sensors".NAV_position.Low_limit_ADC_current := "Sensors".NAV_position.Low_limit_ADC_new;
           "Sensors".NAV_position.High_limit_ADC_current := "Sensors".NAV_position.High_limit_ADC_new;
           "Sensors".NAV_position.Apply := false;
       END_IF;
   ELSE
       "Sensors".NAV_position.Apply := false;
   END_IF;

   (*Положение направл. аппарата дымососа*)
   IF "Sensors".NAD_position.Enable THEN
       "Read_sensor_4_20"(N_module := "Sensors".NAD_position.N_module,
                          N_chanel := "Sensors".NAD_position.N_chanel,
                          Low_limit_phisical_current := "Sensors".NAD_position.Low_limit_phisical_current,
                          High_limit_phisical_current := "Sensors".NAD_position.High_limit_phisical_current,
                          Low_limit_ADC_current := "Sensors".NAD_position.Low_limit_ADC_current,
                          High_limit_ADC_current := "Sensors".NAD_position.High_limit_ADC_current,
                          Current_ADC => "Sensors".NAD_position.Current_ADC,
                          Value => "Sensors".NAD_position.Value,
                          Alarm_sensor => "Sensors".NAD_position.Alarm_sensor,
                          Current => "Sensors".NAD_position.Current);
       //применение изменений значений точек для пересчета сигнала
       IF "Sensors".NAD_position.Apply THEN
           "Sensors".NAD_position.Low_limit_phisical_current := "Sensors".NAD_position.Low_limit_phisical_new;
           "Sensors".NAD_position.High_limit_phisical_current := "Sensors".NAD_position.High_limit_phisical_new;
           "Sensors".NAD_position.Low_limit_ADC_current := "Sensors".NAD_position.Low_limit_ADC_new;
           "Sensors".NAD_position.High_limit_ADC_current := "Sensors".NAD_position.High_limit_ADC_new;
           "Sensors".NAD_position.Apply := false;
       END_IF;
   ELSE
       "Sensors".NAD_position.Apply := false;
   END_IF;

   (*Текущ. значение ПЧ ДВ*)
   IF "Sensors".DV_current_frequency.Enable THEN
       "Read_sensor_4_20"(N_module := "Sensors".DV_current_frequency.N_module,
                          N_chanel := "Sensors".DV_current_frequency.N_chanel,
                          Low_limit_phisical_current := "Sensors".DV_current_frequency.Low_limit_phisical_current,
                          High_limit_phisical_current := "Sensors".DV_current_frequency.High_limit_phisical_current,
                          Low_limit_ADC_current := "Sensors".DV_current_frequency.Low_limit_ADC_current,
                          High_limit_ADC_current := "Sensors".DV_current_frequency.High_limit_ADC_current,
                          Current_ADC => "Sensors".DV_current_frequency.Current_ADC,
                          Value => "Sensors".DV_current_frequency.Value,
                          Alarm_sensor => "Sensors".DV_current_frequency.Alarm_sensor,
                          Current => "Sensors".DV_current_frequency.Current);
       //применение изменений значений точек для пересчета сигнала
       IF "Sensors".DV_current_frequency.Apply THEN
           "Sensors".DV_current_frequency.Low_limit_phisical_current := "Sensors".DV_current_frequency.Low_limit_phisical_new;
           "Sensors".DV_current_frequency.High_limit_phisical_current := "Sensors".DV_current_frequency.High_limit_phisical_new;
           "Sensors".DV_current_frequency.Low_limit_ADC_current := "Sensors".DV_current_frequency.Low_limit_ADC_new;
           "Sensors".DV_current_frequency.High_limit_ADC_current := "Sensors".DV_current_frequency.High_limit_ADC_new;
           "Sensors".DV_current_frequency.Apply := false;
       END_IF;
   ELSE
       "Sensors".DV_current_frequency.Apply := false;
   END_IF;

   (*Текущ. значение ПЧ ДС*)
   IF "Sensors".DS_current_frequency.Enable THEN
       "Read_sensor_4_20"(N_module := "Sensors".DS_current_frequency.N_module,
                          N_chanel := "Sensors".DS_current_frequency.N_chanel,
                          Low_limit_phisical_current := "Sensors".DS_current_frequency.Low_limit_phisical_current,
                          High_limit_phisical_current := "Sensors".DS_current_frequency.High_limit_phisical_current,
                          Low_limit_ADC_current := "Sensors".DS_current_frequency.Low_limit_ADC_current,
                          High_limit_ADC_current := "Sensors".DS_current_frequency.High_limit_ADC_current,
                          Current_ADC => "Sensors".DS_current_frequency.Current_ADC,
                          Value => "Sensors".DS_current_frequency.Value,
                          Alarm_sensor => "Sensors".DS_current_frequency.Alarm_sensor,
                          Current => "Sensors".DS_current_frequency.Current);
       //применение изменений значений точек для пересчета сигнала
       IF "Sensors".DS_current_frequency.Apply THEN
           "Sensors".DS_current_frequency.Low_limit_phisical_current := "Sensors".DS_current_frequency.Low_limit_phisical_new;
           "Sensors".DS_current_frequency.High_limit_phisical_current := "Sensors".DS_current_frequency.High_limit_phisical_new;
           "Sensors".DS_current_frequency.Low_limit_ADC_current := "Sensors".DS_current_frequency.Low_limit_ADC_new;
           "Sensors".DS_current_frequency.High_limit_ADC_current := "Sensors".DS_current_frequency.High_limit_ADC_new;
           "Sensors".DS_current_frequency.Apply := false;
       END_IF;
   ELSE
       "Sensors".DS_current_frequency.Apply := false;
   END_IF;

   (*Температура газа перед БГ*)
   IF "Sensors".T_gas_before_BG.Enable THEN
       "Read_sensor_4_20"(N_module := "Sensors".T_gas_before_BG.N_module,
                          N_chanel := "Sensors".T_gas_before_BG.N_chanel,
                          Low_limit_phisical_current := "Sensors".T_gas_before_BG.Low_limit_phisical_current,
                          High_limit_phisical_current := "Sensors".T_gas_before_BG.High_limit_phisical_current,
                          Low_limit_ADC_current := "Sensors".T_gas_before_BG.Low_limit_ADC_current,
                          High_limit_ADC_current := "Sensors".T_gas_before_BG.High_limit_ADC_current,
                          Current_ADC => "Sensors".T_gas_before_BG.Current_ADC,
                          Value => "Sensors".T_gas_before_BG.Value,
                          Alarm_sensor => "Sensors".T_gas_before_BG.Alarm_sensor,
                          Current => "Sensors".T_gas_before_BG.Current);
       //применение изменений значений точек для пересчета сигнала
       IF "Sensors".T_gas_before_BG.Apply THEN
           "Sensors".T_gas_before_BG.Low_limit_phisical_current := "Sensors".T_gas_before_BG.Low_limit_phisical_new;
           "Sensors".T_gas_before_BG.High_limit_phisical_current := "Sensors".T_gas_before_BG.High_limit_phisical_new;
           "Sensors".T_gas_before_BG.Low_limit_ADC_current := "Sensors".T_gas_before_BG.Low_limit_ADC_new;
           "Sensors".T_gas_before_BG.High_limit_ADC_current := "Sensors".T_gas_before_BG.High_limit_ADC_new;
           "Sensors".T_gas_before_BG.Apply := false;
       END_IF;
   ELSE
       "Sensors".T_gas_before_BG.Apply := false;
   END_IF;

   (*Давление газа перед БГ*)
   IF "Sensors".P_gas_before_BG.Enable THEN
       "Read_sensor_4_20"(N_module := "Sensors".P_gas_before_BG.N_module,
                          N_chanel := "Sensors".P_gas_before_BG.N_chanel,
                          Low_limit_phisical_current := "Sensors".P_gas_before_BG.Low_limit_phisical_current,
                          High_limit_phisical_current := "Sensors".P_gas_before_BG.High_limit_phisical_current,
                          Low_limit_ADC_current := "Sensors".P_gas_before_BG.Low_limit_ADC_current,
                          High_limit_ADC_current := "Sensors".P_gas_before_BG.High_limit_ADC_current,
                          Current_ADC => "Sensors".P_gas_before_BG.Current_ADC,
                          Value => "Sensors".P_gas_before_BG.Value,
                          Alarm_sensor => "Sensors".P_gas_before_BG.Alarm_sensor,
                          Current => "Sensors".P_gas_before_BG.Current);
       //применение изменений значений точек для пересчета сигнала
       IF "Sensors".P_gas_before_BG.Apply THEN
           "Sensors".P_gas_before_BG.Low_limit_phisical_current := "Sensors".P_gas_before_BG.Low_limit_phisical_new;
           "Sensors".P_gas_before_BG.High_limit_phisical_current := "Sensors".P_gas_before_BG.High_limit_phisical_new;
           "Sensors".P_gas_before_BG.Low_limit_ADC_current := "Sensors".P_gas_before_BG.Low_limit_ADC_new;
           "Sensors".P_gas_before_BG.High_limit_ADC_current := "Sensors".P_gas_before_BG.High_limit_ADC_new;
           "Sensors".P_gas_before_BG.Apply := false;
       END_IF;
   ELSE
       "Sensors".P_gas_before_BG.Apply := false;
   END_IF;


   (*Чтение дискретных входов*)
   (*Наличие пламени горелки*)
   IF "Sensors".Burner_flame.Enable THEN
       "Read_discret_signal"(N_module := "Sensors".Burner_flame.N_module,
                             N_chanel := "Sensors".Burner_flame.N_chanel,
                             Invert := "Sensors".Burner_flame.Invert,
                             Value => "Sensors".Burner_flame.Value);
   ELSE
       "Sensors".Burner_flame.Value := false;
   END_IF;

   (*Наличие пламени запальника горелки*)
   IF "Sensors".Igniter_flame.Enable THEN
       "Read_discret_signal"(N_module := "Sensors".Igniter_flame.N_module,
                             N_chanel := "Sensors".Igniter_flame.N_chanel,
                             Invert := "Sensors".Igniter_flame.Invert,
                             Value => "Sensors".Igniter_flame.Value);
   ELSE
       "Sensors".Igniter_flame.Value := false;
   END_IF;

   (*Клапан безопасности закрыт*)
   IF "Sensors".KB_close.Enable THEN
       "Read_discret_signal"(N_module := "Sensors".KB_close.N_module,
                             N_chanel := "Sensors".KB_close.N_chanel,
                             Invert := "Sensors".KB_close.Invert,
                             Value => "Sensors".KB_close.Value);
   ELSE
       "Sensors".KB_close.Value := false;
   END_IF;

   (*Клапан опрессовки открыт*)
   IF "Sensors".KO_open.Enable THEN
       "Read_discret_signal"(N_module := "Sensors".KO_open.N_module,
                             N_chanel := "Sensors".KO_open.N_chanel,
                             Invert := "Sensors".KO_open.Invert,
                             Value => "Sensors".KO_open.Value);
   ELSE
       "Sensors".KO_open.Value := false;
   END_IF;

   (*Клапан запальника открыт*)
   IF "Sensors".KZ_open.Enable THEN
       "Read_discret_signal"(N_module := "Sensors".KZ_open.N_module,
                             N_chanel := "Sensors".KZ_open.N_chanel,
                             Invert := "Sensors".KZ_open.Invert,
                             Value => "Sensors".KZ_open.Value);
   ELSE
       "Sensors".KZ_open.Value := false;
   END_IF;

   (*ПЗК-1 горелки открыт*)
   IF "Sensors".PZK1_open.Enable THEN
       "Read_discret_signal"(N_module := "Sensors".PZK1_open.N_module,
                             N_chanel := "Sensors".PZK1_open.N_chanel,
                             Invert := "Sensors".PZK1_open.Invert,
                             Value => "Sensors".PZK1_open.Value);
   ELSE
       "Sensors".PZK1_open.Value := false;
   END_IF;

   (*ПЗК-2 горелки не закрыт*)
   IF "Sensors".PZK2_not_close.Enable THEN
       "Read_discret_signal"(N_module := "Sensors".PZK2_not_close.N_module,
                             N_chanel := "Sensors".PZK2_not_close.N_chanel,
                             Invert := "Sensors".PZK2_not_close.Invert,
                             Value => "Sensors".PZK2_not_close.Value);
   ELSE
       "Sensors".PZK2_not_close.Value := false;
   END_IF;

   (*Давление газа перед БГ мин.*)
   IF "Sensors".P_gas_before_BG_min.Enable THEN
       "Read_discret_signal"(N_module := "Sensors".P_gas_before_BG_min.N_module,
                             N_chanel := "Sensors".P_gas_before_BG_min.N_chanel,
                             Invert := "Sensors".P_gas_before_BG_min.Invert,
                             Value => "Sensors".P_gas_before_BG_min.Value);
   ELSE
       "Sensors".P_gas_before_BG_min.Value := false;
   END_IF;

   (*Давление газа перед БГ макс.*)
   IF "Sensors".P_gas_before_BG_max.Enable THEN
       "Read_discret_signal"(N_module := "Sensors".P_gas_before_BG_max.N_module,
                             N_chanel := "Sensors".P_gas_before_BG_max.N_chanel,
                             Invert := "Sensors".P_gas_before_BG_max.Invert,
                             Value => "Sensors".P_gas_before_BG_max.Value);
   ELSE
       "Sensors".P_gas_before_BG_max.Value := false;
   END_IF;

   (*Давление воздуха перед горелкой мин.*)
   IF "Sensors".P_air_before_burner_min.Enable THEN
       "Read_discret_signal"(N_module := "Sensors".P_air_before_burner_min.N_module,
                             N_chanel := "Sensors".P_air_before_burner_min.N_chanel,
                             Invert := "Sensors".P_air_before_burner_min.Invert,
                             Value => "Sensors".P_air_before_burner_min.Value);
   ELSE
       "Sensors".P_air_before_burner_min.Value := false;
   END_IF;

   (*Давление газа перед горелкой мин.*)
   IF "Sensors".P_gas_before_burner_min.Enable THEN
       "Read_discret_signal"(N_module := "Sensors".P_gas_before_burner_min.N_module,
                             N_chanel := "Sensors".P_gas_before_burner_min.N_chanel,
                             Invert := "Sensors".P_gas_before_burner_min.Invert,
                             Value => "Sensors".P_gas_before_burner_min.Value);
   ELSE
       "Sensors".P_gas_before_burner_min.Value := false;
   END_IF;

   (*Давление газа перед горелкой макс.*)
   IF "Sensors".P_gas_before_burner_max.Enable THEN
       "Read_discret_signal"(N_module := "Sensors".P_gas_before_burner_max.N_module,
                             N_chanel := "Sensors".P_gas_before_burner_max.N_chanel,
                             Invert := "Sensors".P_gas_before_burner_max.Invert,
                             Value => "Sensors".P_gas_before_burner_max.Value);
   ELSE
       "Sensors".P_gas_before_burner_max.Value := false;
   END_IF;

   (*Регулирующая заслонка газа. открыта*)
   IF "Sensors".ZRG_open.Enable THEN
       "Read_discret_signal"(N_module := "Sensors".ZRG_open.N_module,
                             N_chanel := "Sensors".ZRG_open.N_chanel,
                             Invert := "Sensors".ZRG_open.Invert,
                             Value => "Sensors".ZRG_open.Value);
   ELSE
       "Sensors".ZRG_open.Value := false;
   END_IF;

   (*Регулирующая заслонка газа. закрыта*)
   IF "Sensors".ZRG_close.Enable THEN
       "Read_discret_signal"(N_module := "Sensors".ZRG_close.N_module,
                             N_chanel := "Sensors".ZRG_close.N_chanel,
                             Invert := "Sensors".ZRG_close.Invert,
                             Value => "Sensors".ZRG_close.Value);
   ELSE
       "Sensors".ZRG_close.Value := false;
   END_IF;

   (*Регулирующая заслонка газа. среднее*)
   IF "Sensors".ZRG_middle.Enable THEN
       "Read_discret_signal"(N_module := "Sensors".ZRG_middle.N_module,
                             N_chanel := "Sensors".ZRG_middle.N_chanel,
                             Invert := "Sensors".ZRG_middle.Invert,
                             Value => "Sensors".ZRG_middle.Value);
   ELSE
       "Sensors".ZRG_middle.Value := false;
   END_IF;

   (*Регулирующая заслонка газа. БРУ в положении "Авт"*)
   IF "Sensors".ZRG_avto.Enable THEN
       "Read_discret_signal"(N_module := "Sensors".ZRG_avto.N_module,
                             N_chanel := "Sensors".ZRG_avto.N_chanel,
                             Invert := "Sensors".ZRG_avto.Invert,
                             Value => "Sensors".ZRG_avto.Value);
   ELSE
       "Sensors".ZRG_avto.Value := false;
   END_IF;

   (*Регулирующая заслонка НАВ. открыта*)
   IF "Sensors".NAV_open.Enable THEN
       "Read_discret_signal"(N_module := "Sensors".NAV_open.N_module,
                             N_chanel := "Sensors".NAV_open.N_chanel,
                             Invert := "Sensors".NAV_open.Invert,
                             Value => "Sensors".NAV_open.Value);
   ELSE
       "Sensors".NAV_open.Value := false;
   END_IF;

   (*Регулирующая заслонка НАВ. закрыта*)
   IF "Sensors".NAV_close.Enable THEN
       "Read_discret_signal"(N_module := "Sensors".NAV_close.N_module,
                             N_chanel := "Sensors".NAV_close.N_chanel,
                             Invert := "Sensors".NAV_close.Invert,
                             Value => "Sensors".NAV_close.Value);
   ELSE
       "Sensors".NAV_close.Value := false;
   END_IF;

   (*Регулирующая заслонка НАВ. среднее*)
   IF "Sensors".NAV_middle.Enable THEN
       "Read_discret_signal"(N_module := "Sensors".NAV_middle.N_module,
                             N_chanel := "Sensors".NAV_middle.N_chanel,
                             Invert := "Sensors".NAV_middle.Invert,
                             Value => "Sensors".NAV_middle.Value);
   ELSE
       "Sensors".NAV_middle.Value := false;
   END_IF;

   (*Регулирующая заслонка НАВ. БРУ в положении "Авт"*)
   IF "Sensors".NAV_avto.Enable THEN
       "Read_discret_signal"(N_module := "Sensors".NAV_avto.N_module,
                             N_chanel := "Sensors".NAV_avto.N_chanel,
                             Invert := "Sensors".NAV_avto.Invert,
                             Value => "Sensors".NAV_avto.Value);
   ELSE
       "Sensors".NAV_avto.Value := false;
   END_IF;

   (*Регулирующая заслонка НАД. открыта*)
   IF "Sensors".NAD_open.Enable THEN
       "Read_discret_signal"(N_module := "Sensors".NAD_open.N_module,
                             N_chanel := "Sensors".NAD_open.N_chanel,
                             Invert := "Sensors".NAD_open.Invert,
                             Value => "Sensors".NAD_open.Value);
   ELSE
       "Sensors".NAD_open.Value := false;
   END_IF;

   (*Регулирующая заслонка НАД. закрыта*)
   IF "Sensors".NAD_close.Enable THEN
       "Read_discret_signal"(N_module := "Sensors".NAD_close.N_module,
                             N_chanel := "Sensors".NAD_close.N_chanel,
                             Invert := "Sensors".NAD_close.Invert,
                             Value => "Sensors".NAD_close.Value);
   ELSE
       "Sensors".NAD_close.Value := false;
   END_IF;

   (*Регулирующая заслонка НАД. среднее*)
   IF "Sensors".NAD_middle.Enable THEN
       "Read_discret_signal"(N_module := "Sensors".NAD_middle.N_module,
                             N_chanel := "Sensors".NAD_middle.N_chanel,
                             Invert := "Sensors".NAD_middle.Invert,
                             Value => "Sensors".NAD_middle.Value);
   ELSE
       "Sensors".NAD_middle.Value := false;
   END_IF;

   (*Регулирующая заслонка НАД. БРУ в положении "Авт"*)
   IF "Sensors".NAD_avto.Enable THEN
       "Read_discret_signal"(N_module := "Sensors".NAD_avto.N_module,
                             N_chanel := "Sensors".NAD_avto.N_chanel,
                             Invert := "Sensors".NAD_avto.Invert,
                             Value => "Sensors".NAD_avto.Value);
   ELSE
       "Sensors".NAD_avto.Value := false;
   END_IF;

   (*Разрежение в топке котла мин.*)
   IF "Sensors".dP_furnace_boiler_min.Enable THEN
       "Read_discret_signal"(N_module := "Sensors".dP_furnace_boiler_min.N_module,
                             N_chanel := "Sensors".dP_furnace_boiler_min.N_chanel,
                             Invert := "Sensors".dP_furnace_boiler_min.Invert,
                             Value => "Sensors".dP_furnace_boiler_min.Value);
   ELSE
       "Sensors".dP_furnace_boiler_min.Value := false;
   END_IF;

   (*Температура сетевой воды после котла макс.*)
   IF "Sensors".T_water_after_boiler_max.Enable THEN
       "Read_discret_signal"(N_module := "Sensors".T_water_after_boiler_max.N_module,
                             N_chanel := "Sensors".T_water_after_boiler_max.N_chanel,
                             Invert := "Sensors".T_water_after_boiler_max.Invert,
                             Value => "Sensors".T_water_after_boiler_max.Value);
   ELSE
       "Sensors".T_water_after_boiler_max.Value := false;
   END_IF;

   (*Расход сетевой воды через котел мин.*)
   IF "Sensors".Q_water_boiler_min.Enable THEN
       "Read_discret_signal"(N_module := "Sensors".Q_water_boiler_min.N_module,
                             N_chanel := "Sensors".Q_water_boiler_min.N_chanel,
                             Invert := "Sensors".Q_water_boiler_min.Invert,
                             Value => "Sensors".Q_water_boiler_min.Value);
   ELSE
       "Sensors".Q_water_boiler_min.Value := false;
   END_IF;

   (*Расход сетевой воды через котел макс.*)
   IF "Sensors".Q_water_boiler_max.Enable THEN
       "Read_discret_signal"(N_module := "Sensors".Q_water_boiler_max.N_module,
                             N_chanel := "Sensors".Q_water_boiler_max.N_chanel,
                             Invert := "Sensors".Q_water_boiler_max.Invert,
                             Value => "Sensors".Q_water_boiler_max.Value);
   ELSE
       "Sensors".Q_water_boiler_max.Value := false;
   END_IF;

   (*Давление сетевой воды после котла мин.*)
   IF "Sensors".P_water_after_boiler_min.Enable THEN
       "Read_discret_signal"(N_module := "Sensors".P_water_after_boiler_min.N_module,
                             N_chanel := "Sensors".P_water_after_boiler_min.N_chanel,
                             Invert := "Sensors".P_water_after_boiler_min.Invert,
                             Value => "Sensors".P_water_after_boiler_min.Value);
   ELSE
       "Sensors".P_water_after_boiler_min.Value := false;
   END_IF;

   (*Давление сетевой воды после котла макс.*)
   IF "Sensors".P_water_after_boiler_max.Enable THEN
       "Read_discret_signal"(N_module := "Sensors".P_water_after_boiler_max.N_module,
                             N_chanel := "Sensors".P_water_after_boiler_max.N_chanel,
                             Invert := "Sensors".P_water_after_boiler_max.Invert,
                             Value => "Sensors".P_water_after_boiler_max.Value);
   ELSE
       "Sensors".P_water_after_boiler_max.Value := false;
   END_IF;

   (*Давление сетевой воды перед котлом мин.*)
   IF "Sensors".P_water_before_boiler_min.Enable THEN
       "Read_discret_signal"(N_module := "Sensors".P_water_before_boiler_min.N_module,
                             N_chanel := "Sensors".P_water_before_boiler_min.N_chanel,
                             Invert := "Sensors".P_water_before_boiler_min.Invert,
                             Value => "Sensors".P_water_before_boiler_min.Value);
   ELSE
       "Sensors".P_water_before_boiler_min.Value := false;
   END_IF;

   (*Давление сетевой воды перед котлом макс.*)
   IF "Sensors".P_water_before_boiler_max.Enable THEN
       "Read_discret_signal"(N_module := "Sensors".P_water_before_boiler_max.N_module,
                             N_chanel := "Sensors".P_water_before_boiler_max.N_chanel,
                             Invert := "Sensors".P_water_before_boiler_max.Invert,
                             Value => "Sensors".P_water_before_boiler_max.Value);
   ELSE
       "Sensors".P_water_before_boiler_max.Value := false;
   END_IF;

   (*Вызов к шакафу электропитания*)
   IF "Sensors".Call_power_supply_сabinet.Enable THEN
       "Read_discret_signal"(N_module := "Sensors".Call_power_supply_сabinet.N_module,
                             N_chanel := "Sensors".Call_power_supply_сabinet.N_chanel,
                             Invert := "Sensors".Call_power_supply_сabinet.Invert,
                             Value => "Sensors".Call_power_supply_сabinet.Value);
   ELSE
       "Sensors".Call_power_supply_сabinet.Value := false;
   END_IF;

   (*Авария ПЧ ДВ*)
   IF "Sensors".DV_Invertor_alarm.Enable THEN
       "Read_discret_signal"(N_module := "Sensors".DV_Invertor_alarm.N_module,
                             N_chanel := "Sensors".DV_Invertor_alarm.N_chanel,
                             Invert := "Sensors".DV_Invertor_alarm.Invert,
                             Value => "Sensors".DV_Invertor_alarm.Value);
   ELSE
       "Sensors".DV_Invertor_alarm.Value := false;
   END_IF;

   (*Управление «Местный» ДВ*)
   IF "Sensors".DV_local_control.Enable THEN
       "Read_discret_signal"(N_module := "Sensors".DV_local_control.N_module,
                             N_chanel := "Sensors".DV_local_control.N_chanel,
                             Invert := "Sensors".DV_local_control.Invert,
                             Value => "Sensors".DV_local_control.Value);
   ELSE
       "Sensors".DV_local_control.Value := false;
   END_IF;

   (*Управление «Дистанционный» ДВ*)
   IF "Sensors".DV_dist_control.Enable THEN
       "Read_discret_signal"(N_module := "Sensors".DV_dist_control.N_module,
                             N_chanel := "Sensors".DV_dist_control.N_chanel,
                             Invert := "Sensors".DV_dist_control.Invert,
                             Value => "Sensors".DV_dist_control.Value);
   ELSE
       "Sensors".DV_dist_control.Value := false;
   END_IF;

   (*Режим "СЕТЬ" ДВ*)
   IF "Sensors".DV_powergrid_mode.Enable THEN
       "Read_discret_signal"(N_module := "Sensors".DV_powergrid_mode.N_module,
                             N_chanel := "Sensors".DV_powergrid_mode.N_chanel,
                             Invert := "Sensors".DV_powergrid_mode.Invert,
                             Value => "Sensors".DV_powergrid_mode.Value);
   ELSE
       "Sensors".DV_powergrid_mode.Value := false;
   END_IF;

   (*Режим "ПЧ" ДВ*)
   IF "Sensors".DV_invertor_mode.Enable THEN
       "Read_discret_signal"(N_module := "Sensors".DV_invertor_mode.N_module,
                             N_chanel := "Sensors".DV_invertor_mode.N_chanel,
                             Invert := "Sensors".DV_invertor_mode.Invert,
                             Value => "Sensors".DV_invertor_mode.Value);
   ELSE
       "Sensors".DV_invertor_mode.Value := false;
   END_IF;

   (*Автомат работы ДВ от ПЧ включен*)
   IF "Sensors".DV_invertor_QF_on.Enable THEN
       "Read_discret_signal"(N_module := "Sensors".DV_invertor_QF_on.N_module,
                             N_chanel := "Sensors".DV_invertor_QF_on.N_chanel,
                             Invert := "Sensors".DV_invertor_QF_on.Invert,
                             Value => "Sensors".DV_invertor_QF_on.Value);
   ELSE
       "Sensors".DV_invertor_QF_on.Value := false;
   END_IF;

   (*Автомат работы ДВ от сети включен*)
   IF "Sensors".DV_powergrid_QF_on.Enable THEN
       "Read_discret_signal"(N_module := "Sensors".DV_powergrid_QF_on.N_module,
                             N_chanel := "Sensors".DV_powergrid_QF_on.N_chanel,
                             Invert := "Sensors".DV_powergrid_QF_on.Invert,
                             Value => "Sensors".DV_powergrid_QF_on.Value);
   ELSE
       "Sensors".DV_powergrid_QF_on.Value := false;
   END_IF;

   (*Включен ДВ от ПЧ*)
   IF "Sensors".DV_invertor_on.Enable THEN
       "Read_discret_signal"(N_module := "Sensors".DV_invertor_on.N_module,
                             N_chanel := "Sensors".DV_invertor_on.N_chanel,
                             Invert := "Sensors".DV_invertor_on.Invert,
                             Value => "Sensors".DV_invertor_on.Value);
   ELSE
       "Sensors".DV_invertor_on.Value := false;
   END_IF;

   (*Включен ДВ от сети*)
   IF "Sensors".DV_powergrid_on.Enable THEN
       "Read_discret_signal"(N_module := "Sensors".DV_powergrid_on.N_module,
                             N_chanel := "Sensors".DV_powergrid_on.N_chanel,
                             Invert := "Sensors".DV_powergrid_on.Invert,
                             Value => "Sensors".DV_powergrid_on.Value);
   ELSE
       "Sensors".DV_powergrid_on.Value := false;
   END_IF;

   (*Нет напряжения сети ШУД ДВ*)
   IF "Sensors".DV_no_voltage.Enable THEN
       "Read_discret_signal"(N_module := "Sensors".DV_no_voltage.N_module,
                             N_chanel := "Sensors".DV_no_voltage.N_chanel,
                             Invert := "Sensors".DV_no_voltage.Invert,
                             Value => "Sensors".DV_no_voltage.Value);
   ELSE
       "Sensors".DV_no_voltage.Value := false;
   END_IF;

   (*Авария ПЧ ДС*)
   IF "Sensors".DS_Invertor_alarm.Enable THEN
       "Read_discret_signal"(N_module := "Sensors".DS_Invertor_alarm.N_module,
                             N_chanel := "Sensors".DS_Invertor_alarm.N_chanel,
                             Invert := "Sensors".DS_Invertor_alarm.Invert,
                             Value => "Sensors".DS_Invertor_alarm.Value);
   ELSE
       "Sensors".DS_Invertor_alarm.Value := false;
   END_IF;

   (*Управление «Местный» ДС*)
   IF "Sensors".DS_local_control.Enable THEN
       "Read_discret_signal"(N_module := "Sensors".DS_local_control.N_module,
                             N_chanel := "Sensors".DS_local_control.N_chanel,
                             Invert := "Sensors".DS_local_control.Invert,
                             Value => "Sensors".DS_local_control.Value);
   ELSE
       "Sensors".DS_local_control.Value := false;
   END_IF;

   (*Управление «Дистанционный» ДС*)
   IF "Sensors".DS_dist_control.Enable THEN
       "Read_discret_signal"(N_module := "Sensors".DS_dist_control.N_module,
                             N_chanel := "Sensors".DS_dist_control.N_chanel,
                             Invert := "Sensors".DS_dist_control.Invert,
                             Value => "Sensors".DS_dist_control.Value);
   ELSE
       "Sensors".DS_dist_control.Value := false;
   END_IF;

   (*Режим "СЕТЬ" ДС*)
   IF "Sensors".DS_powergrid_mode.Enable THEN
       "Read_discret_signal"(N_module := "Sensors".DS_powergrid_mode.N_module,
                             N_chanel := "Sensors".DS_powergrid_mode.N_chanel,
                             Invert := "Sensors".DS_powergrid_mode.Invert,
                             Value => "Sensors".DS_powergrid_mode.Value);
   ELSE
       "Sensors".DS_powergrid_mode.Value := false;
   END_IF;

   (*Режим "ПЧ" ДС*)
   IF "Sensors".DS_invertor_mode.Enable THEN
       "Read_discret_signal"(N_module := "Sensors".DS_invertor_mode.N_module,
                             N_chanel := "Sensors".DS_invertor_mode.N_chanel,
                             Invert := "Sensors".DS_invertor_mode.Invert,
                             Value => "Sensors".DS_invertor_mode.Value);
   ELSE
       "Sensors".DS_invertor_mode.Value := false;
   END_IF;

   (*Автомат работы ДС от ПЧ включен*)
   IF "Sensors".DS_invertor_QF_on.Enable THEN
       "Read_discret_signal"(N_module := "Sensors".DS_invertor_QF_on.N_module,
                             N_chanel := "Sensors".DS_invertor_QF_on.N_chanel,
                             Invert := "Sensors".DS_invertor_QF_on.Invert,
                             Value => "Sensors".DS_invertor_QF_on.Value);
   ELSE
       "Sensors".DS_invertor_QF_on.Value := false;
   END_IF;

   (*Автомат работы ДС от сети включен*)
   IF "Sensors".DS_powergrid_QF_on.Enable THEN
       "Read_discret_signal"(N_module := "Sensors".DS_powergrid_QF_on.N_module,
                             N_chanel := "Sensors".DS_powergrid_QF_on.N_chanel,
                             Invert := "Sensors".DS_powergrid_QF_on.Invert,
                             Value => "Sensors".DS_powergrid_QF_on.Value);
   ELSE
       "Sensors".DS_powergrid_QF_on.Value := false;
   END_IF;

   (*ДС включен от ПЧ*)
   IF "Sensors".DS_invertor_on.Enable THEN
       "Read_discret_signal"(N_module := "Sensors".DS_invertor_on.N_module,
                             N_chanel := "Sensors".DS_invertor_on.N_chanel,
                             Invert := "Sensors".DS_invertor_on.Invert,
                             Value => "Sensors".DS_invertor_on.Value);
   ELSE
       "Sensors".DS_invertor_on.Value := false;
   END_IF;

   (*ДС включен от сети*)
   IF "Sensors".DS_powergrid_on.Enable THEN
       "Read_discret_signal"(N_module := "Sensors".DS_powergrid_on.N_module,
                             N_chanel := "Sensors".DS_powergrid_on.N_chanel,
                             Invert := "Sensors".DS_powergrid_on.Invert,
                             Value => "Sensors".DS_powergrid_on.Value);
   ELSE
       "Sensors".DS_powergrid_on.Value := false;
   END_IF;

   (*Нет напряжения сети ШУД ДС*)
   IF "Sensors".DS_no_voltage.Enable THEN
       "Read_discret_signal"(N_module := "Sensors".DS_no_voltage.N_module,
                             N_chanel := "Sensors".DS_no_voltage.N_chanel,
                             Invert := "Sensors".DS_no_voltage.Invert,
                             Value => "Sensors".DS_no_voltage.Value);
   ELSE
       "Sensors".DS_no_voltage.Value := false;
   END_IF;

   (*Загазованность СО I порог*)
   IF "Sensors".CO_1.Enable THEN
       "Read_discret_signal"(N_module := "Sensors".CO_1.N_module,
                             N_chanel := "Sensors".CO_1.N_chanel,
                             Invert := "Sensors".CO_1.Invert,
                             Value => "Sensors".CO_1.Value);
   ELSE
       "Sensors".CO_1.Value := false;
   END_IF;

   (*Загазованность СО II порог*)
   IF "Sensors".CO_2.Enable THEN
       "Read_discret_signal"(N_module := "Sensors".CO_2.N_module,
                             N_chanel := "Sensors".CO_2.N_chanel,
                             Invert := "Sensors".CO_2.Invert,
                             Value => "Sensors".CO_2.Value);
   ELSE
       "Sensors".CO_2.Value := false;
   END_IF;

   (*Загазованность CH4 порог*)
   IF "Sensors".CH4.Enable THEN
       "Read_discret_signal"(N_module := "Sensors".CH4.N_module,
                             N_chanel := "Sensors".CH4.N_chanel,
                             Invert := "Sensors".CH4.Invert,
                             Value => "Sensors".CH4.Value);
   ELSE
       "Sensors".CH4.Value := false;
   END_IF;

   (*Кнопка СТОП*)
   IF "Sensors".Btn_STOP.Enable THEN
       "Read_discret_signal"(N_module := "Sensors".Btn_STOP.N_module,
                             N_chanel := "Sensors".Btn_STOP.N_chanel,
                             Invert := "Sensors".Btn_STOP.Invert,
                             Value => "Sensors".Btn_STOP.Value);
   ELSE
       "Sensors".Btn_STOP.Value := false;
   END_IF;

   (*Кнопка Вентиляция*)
   IF "Sensors".Btn_Ventilation.Enable THEN
       "Read_discret_signal"(N_module := "Sensors".Btn_Ventilation.N_module,
                             N_chanel := "Sensors".Btn_Ventilation.N_chanel,
                             Invert := "Sensors".Btn_Ventilation.Invert,
                             Value => "Sensors".Btn_Ventilation.Value);
   ELSE
       "Sensors".Btn_Ventilation.Value := false;
   END_IF;

   (*Кнопка Розжиг*)
   IF "Sensors".Btn_Ignition.Enable THEN
       "Read_discret_signal"(N_module := "Sensors".Btn_Ignition.N_module,
                             N_chanel := "Sensors".Btn_Ignition.N_chanel,
                             Invert := "Sensors".Btn_Ignition.Invert,
                             Value => "Sensors".Btn_Ignition.Value);
   ELSE
       "Sensors".Btn_Ignition.Value := false;
   END_IF;

   (*Кнопка Сброс звука / Проверка звука*)
   IF "Sensors".Btn_Sound.Enable THEN
       "Read_discret_signal"(N_module := "Sensors".Btn_Sound.N_module,
                             N_chanel := "Sensors".Btn_Sound.N_chanel,
                             Invert := "Sensors".Btn_Sound.Invert,
                             Value => "Sensors".Btn_Sound.Value);
   ELSE
       "Sensors".Btn_Sound.Value := false;
   END_IF;

   (*Контроль питания сети ~400В 1ШЭУ*)
   IF "Sensors".SHEU_voltage_ok.Enable THEN
       "Read_discret_signal"(N_module := "Sensors".SHEU_voltage_ok.N_module,
                             N_chanel := "Sensors".SHEU_voltage_ok.N_chanel,
                             Invert := "Sensors".SHEU_voltage_ok.Invert,
                             Value => "Sensors".SHEU_voltage_ok.Value);
   ELSE
       "Sensors".SHEU_voltage_ok.Value := false;
   END_IF;

   (*ПЗК-2 горелки открыт*)
   IF "Sensors".PZK2_open.Enable THEN
       "Read_discret_signal"(N_module := "Sensors".PZK2_open.N_module,
                             N_chanel := "Sensors".PZK2_open.N_chanel,
                             Invert := "Sensors".PZK2_open.Invert,
                             Value => "Sensors".PZK2_open.Value);
   ELSE
       "Sensors".PZK2_open.Value := false;
   END_IF;

   (*Питание контроллера от ИБП*)
   IF "Sensors".Power_PLC_from_UPS.Enable THEN
       "Read_discret_signal"(N_module := "Sensors".Power_PLC_from_UPS.N_module,
                             N_chanel := "Sensors".Power_PLC_from_UPS.N_chanel,
                             Invert := "Sensors".Power_PLC_from_UPS.Invert,
                             Value => "Sensors".Power_PLC_from_UPS.Value);
   ELSE
       "Sensors".Power_PLC_from_UPS.Value := false;
   END_IF;

   (*Заряд батареи ИБП низкий*)
   IF "Sensors".UPS_Low_charge.Enable THEN
       "Read_discret_signal"(N_module := "Sensors".UPS_Low_charge.N_module,
                             N_chanel := "Sensors".UPS_Low_charge.N_chanel,
                             Invert := "Sensors".UPS_Low_charge.Invert,
                             Value => "Sensors".UPS_Low_charge.Value);
   ELSE
       "Sensors".UPS_Low_charge.Value := false;
   END_IF;

   (*ЗРГ Напряжение в норме*)
   IF "Sensors".ZRG_voltage_ok.Enable THEN
       "Read_discret_signal"(N_module := "Sensors".ZRG_voltage_ok.N_module,
                             N_chanel := "Sensors".ZRG_voltage_ok.N_chanel,
                             Invert := "Sensors".ZRG_voltage_ok.Invert,
                             Value => "Sensors".ZRG_voltage_ok.Value);
   ELSE
       "Sensors".ZRG_voltage_ok.Value := false;
   END_IF;

   (*НАВ Напряжение в норме*)
   IF "Sensors".NAV_voltage_ok.Enable THEN
       "Read_discret_signal"(N_module := "Sensors".NAV_voltage_ok.N_module,
                             N_chanel := "Sensors".NAV_voltage_ok.N_chanel,
                             Invert := "Sensors".NAV_voltage_ok.Invert,
                             Value => "Sensors".NAV_voltage_ok.Value);
   ELSE
       "Sensors".NAV_voltage_ok.Value := false;
   END_IF;

   (*НАД Напряжение в норме*)
   IF "Sensors".NAD_voltage_ok.Enable THEN
       "Read_discret_signal"(N_module := "Sensors".NAD_voltage_ok.N_module,
                             N_chanel := "Sensors".NAD_voltage_ok.N_chanel,
                             Invert := "Sensors".NAD_voltage_ok.Invert,
                             Value => "Sensors".NAD_voltage_ok.Value);
   ELSE
       "Sensors".NAD_voltage_ok.Value := false;
   END_IF;

   (*ЗДГ перед БГ. не открыта*)
   IF "Sensors".ZDG_no_open.Enable THEN
       "Read_discret_signal"(N_module := "Sensors".ZDG_no_open.N_module,
                             N_chanel := "Sensors".ZDG_no_open.N_chanel,
                             Invert := "Sensors".ZDG_no_open.Invert,
                             Value => "Sensors".ZDG_no_open.Value);
   ELSE
       "Sensors".ZDG_no_open.Value := false;
   END_IF;

   (*ЗДГ перед БГ. не закрыта*)
   IF "Sensors".ZDG_no_close.Enable THEN
       "Read_discret_signal"(N_module := "Sensors".ZDG_no_close.N_module,
                             N_chanel := "Sensors".ZDG_no_close.N_chanel,
                             Invert := "Sensors".ZDG_no_close.Invert,
                             Value => "Sensors".ZDG_no_close.Value);
   ELSE
       "Sensors".ZDG_no_close.Value := false;
   END_IF;

   (*ЗДГ перед БГ. ход открытие*)
   IF "Sensors".ZDG_opening.Enable THEN
       "Read_discret_signal"(N_module := "Sensors".ZDG_opening.N_module,
                             N_chanel := "Sensors".ZDG_opening.N_chanel,
                             Invert := "Sensors".ZDG_opening.Invert,
                             Value => "Sensors".ZDG_opening.Value);
   ELSE
       "Sensors".ZDG_opening.Value := false;
   END_IF;

   (*ЗДГ перед БГ. ход закрытие*)
   IF "Sensors".ZDG_closing.Enable THEN
       "Read_discret_signal"(N_module := "Sensors".ZDG_closing.N_module,
                             N_chanel := "Sensors".ZDG_closing.N_chanel,
                             Invert := "Sensors".ZDG_closing.Invert,
                             Value => "Sensors".ZDG_closing.Value);
   ELSE
       "Sensors".ZDG_closing.Value := false;
   END_IF;

   (*ЗДГ перед БГ. Напряжение в норме*)
   IF "Sensors".ZDG_voltage_ok.Enable THEN
       "Read_discret_signal"(N_module := "Sensors".ZDG_voltage_ok.N_module,
                             N_chanel := "Sensors".ZDG_voltage_ok.N_chanel,
                             Invert := "Sensors".ZDG_voltage_ok.Invert,
                             Value => "Sensors".ZDG_voltage_ok.Value);
   ELSE
       "Sensors".ZDG_voltage_ok.Value := false;
   END_IF;

   (*ЗДСВ перед котлом. не открыта*)
   IF "Sensors".ZDSV_before_boiler_no_open.Enable THEN
       "Read_discret_signal"(N_module := "Sensors".ZDSV_before_boiler_no_open.N_module,
                             N_chanel := "Sensors".ZDSV_before_boiler_no_open.N_chanel,
                             Invert := "Sensors".ZDSV_before_boiler_no_open.Invert,
                             Value => "Sensors".ZDSV_before_boiler_no_open.Value);
   ELSE
       "Sensors".ZDSV_before_boiler_no_open.Value := false;
   END_IF;

   (*ЗДСВ перед котлом. не закрыта*)
   IF "Sensors".ZDSV_before_boiler_no_close.Enable THEN
       "Read_discret_signal"(N_module := "Sensors".ZDSV_before_boiler_no_close.N_module,
                             N_chanel := "Sensors".ZDSV_before_boiler_no_close.N_chanel,
                             Invert := "Sensors".ZDSV_before_boiler_no_close.Invert,
                             Value => "Sensors".ZDSV_before_boiler_no_close.Value);
   ELSE
       "Sensors".ZDSV_before_boiler_no_close.Value := false;
   END_IF;

   (*ЗДСВ перед котлом. ход открытие*)
   IF "Sensors".ZDSV_before_boiler_opening.Enable THEN
       "Read_discret_signal"(N_module := "Sensors".ZDSV_before_boiler_opening.N_module,
                             N_chanel := "Sensors".ZDSV_before_boiler_opening.N_chanel,
                             Invert := "Sensors".ZDSV_before_boiler_opening.Invert,
                             Value => "Sensors".ZDSV_before_boiler_opening.Value);
   ELSE
       "Sensors".ZDSV_before_boiler_opening.Value := false;
   END_IF;

   (*ЗДСВ перед котлом. ход закрытие*)
   IF "Sensors".ZDSV_before_boiler_closing.Enable THEN
       "Read_discret_signal"(N_module := "Sensors".ZDSV_before_boiler_closing.N_module,
                             N_chanel := "Sensors".ZDSV_before_boiler_closing.N_chanel,
                             Invert := "Sensors".ZDSV_before_boiler_closing.Invert,
                             Value => "Sensors".ZDSV_before_boiler_closing.Value);
   ELSE
       "Sensors".ZDSV_before_boiler_closing.Value := false;
   END_IF;

   (*ЗДСВ перед котлом. Напряжение в норме*)
   IF "Sensors".ZDSV_before_boiler_voltage_ok.Enable THEN
       "Read_discret_signal"(N_module := "Sensors".ZDSV_before_boiler_voltage_ok.N_module,
                             N_chanel := "Sensors".ZDSV_before_boiler_voltage_ok.N_chanel,
                             Invert := "Sensors".ZDSV_before_boiler_voltage_ok.Invert,
                             Value => "Sensors".ZDSV_before_boiler_voltage_ok.Value);
   ELSE
       "Sensors".ZDSV_before_boiler_voltage_ok.Value := false;
   END_IF;

   (*ЗДСВ перед котлом. ограничитель крутящего момента*)
   IF "Sensors".ZDSV_before_boiler_limit_rotational_moment.Enable THEN
       "Read_discret_signal"(N_module := "Sensors".ZDSV_before_boiler_limit_rotational_moment.N_module,
                             N_chanel := "Sensors".ZDSV_before_boiler_limit_rotational_moment.N_chanel,
                             Invert := "Sensors".ZDSV_before_boiler_limit_rotational_moment.Invert,
                             Value => "Sensors".ZDSV_before_boiler_limit_rotational_moment.Value);
   ELSE
       "Sensors".ZDSV_before_boiler_limit_rotational_moment.Value := false;
   END_IF;

   (*ЗДСВ после котла. не открыта*)
   IF "Sensors".ZDSV_after_boiler_no_open.Enable THEN
       "Read_discret_signal"(N_module := "Sensors".ZDSV_after_boiler_no_open.N_module,
                             N_chanel := "Sensors".ZDSV_after_boiler_no_open.N_chanel,
                             Invert := "Sensors".ZDSV_after_boiler_no_open.Invert,
                             Value => "Sensors".ZDSV_after_boiler_no_open.Value);
   ELSE
       "Sensors".ZDSV_after_boiler_no_open.Value := false;
   END_IF;

   (*ЗДСВ после котла. не закрыта*)
   IF "Sensors".ZDSV_after_boiler_no_close.Enable THEN
       "Read_discret_signal"(N_module := "Sensors".ZDSV_after_boiler_no_close.N_module,
                             N_chanel := "Sensors".ZDSV_after_boiler_no_close.N_chanel,
                             Invert := "Sensors".ZDSV_after_boiler_no_close.Invert,
                             Value => "Sensors".ZDSV_after_boiler_no_close.Value);
   ELSE
       "Sensors".ZDSV_after_boiler_no_close.Value := false;
   END_IF;

   (*ЗДСВ после котла. ход открытие*)
   IF "Sensors".ZDSV_after_boiler_opening.Enable THEN
       "Read_discret_signal"(N_module := "Sensors".ZDSV_after_boiler_opening.N_module,
                             N_chanel := "Sensors".ZDSV_after_boiler_opening.N_chanel,
                             Invert := "Sensors".ZDSV_after_boiler_opening.Invert,
                             Value => "Sensors".ZDSV_after_boiler_opening.Value);
   ELSE
       "Sensors".ZDSV_after_boiler_opening.Value := false;
   END_IF;

   (*ЗДСВ после котла. ход закрытие*)
   IF "Sensors".ZDSV_after_boiler_closing.Enable THEN
       "Read_discret_signal"(N_module := "Sensors".ZDSV_after_boiler_closing.N_module,
                             N_chanel := "Sensors".ZDSV_after_boiler_closing.N_chanel,
                             Invert := "Sensors".ZDSV_after_boiler_closing.Invert,
                             Value => "Sensors".ZDSV_after_boiler_closing.Value);
   ELSE
       "Sensors".ZDSV_after_boiler_closing.Value := false;
   END_IF;

   (*ЗДСВ после котла. Напряжение в норме*)
   IF "Sensors".ZDSV_after_boiler_voltage_ok.Enable THEN
       "Read_discret_signal"(N_module := "Sensors".ZDSV_after_boiler_voltage_ok.N_module,
                             N_chanel := "Sensors".ZDSV_after_boiler_voltage_ok.N_chanel,
                             Invert := "Sensors".ZDSV_after_boiler_voltage_ok.Invert,
                             Value => "Sensors".ZDSV_after_boiler_voltage_ok.Value);
   ELSE
       "Sensors".ZDSV_after_boiler_voltage_ok.Value := false;
   END_IF;

   (*ЗДСВ после котла. ограничитель крутящего момента*)
   IF "Sensors".ZDSV_after_boiler_limit_rotational_moment.Enable THEN
       "Read_discret_signal"(N_module := "Sensors".ZDSV_after_boiler_limit_rotational_moment.N_module,
                             N_chanel := "Sensors".ZDSV_after_boiler_limit_rotational_moment.N_chanel,
                             Invert := "Sensors".ZDSV_after_boiler_limit_rotational_moment.Invert,
                             Value => "Sensors".ZDSV_after_boiler_limit_rotational_moment.Value);
   ELSE
       "Sensors".ZDSV_after_boiler_limit_rotational_moment.Value := false;
   END_IF;


   (*Расчетные параметры*)
   (*Расход сетевой воды через котел (м3/ч)*)
   IF "Sensors".Q_water_boiler.Enable THEN
       "Sensors".Q_water_boiler.Value := ("Sensors".Q_water_boiler."a" * "Sensors".Q_water_boiler.Ksh * "Sensors".Q_water_boiler.Kp * 3.1415926 * SQR("Sensors".Q_water_boiler.d) / 4) * SQRT(2 * "Sensors".dP_water_boiler.Value*1000 / "Sensors".Q_water_boiler.ro) * 3600;
   ELSE
       "Sensors".Q_water_boiler.Value := 0;
   END_IF;

   (*Расход газа (м3/ч)*)
   IF "Sensors".Q_gas.Enable THEN
       (*Расчет относительного диаметра сужающего устройства (в 4 степени)*)
       "Sensors".Q_gas.B4 := ("Sensors".Q_gas.d / "Sensors".Q_gas.Dtrub) ** 4;
       (*Значение Р газа*)
       IF NOT "Sensors".Q_gas.Pgas_fixed_value_on AND "Sensors".P_gas_before_BG.Enable THEN
           "Sensors".Q_gas.Pgas := "Sensors".P_gas_before_BG.Value;
       ELSE
           "Sensors".Q_gas.Pgas := "Sensors".Q_gas.Pgas_fixed_value;
       END_IF;
       (*Значение Т газа*)
       IF NOT "Sensors".Q_gas.Tgas_fixed_value_on AND "Sensors".T_gas_before_BG.Enable THEN
           "Sensors".Q_gas.Tgas := "Sensors".T_gas_before_BG.Value;
       ELSE
           "Sensors".Q_gas.Tgas := "Sensors".Q_gas.Tgas_fixed_value;
       END_IF;

       (*Расчет коэффициента расширения*)
       "Sensors".Q_gas."E" := 1 - ((0.351 + (0.256 * "Sensors".Q_gas.B4) + (0.93 * SQR("Sensors".Q_gas.B4))) * (1 - ((1 - ("Sensors".dP_gas_boiler.Value / "Sensors".Q_gas.Pgas)) ** (1 / 1.3155))));
       //"Sensors".Q_gas.E := 1 - ((0.351 + 0.256 * "Sensors".Q_gas.B4) + (0.93 * SQR("Sensors".Q_gas.B4))) * (1 - (1 - "Sensors".dP_gas_boiler.Value / 141.3232) ** (1 / 1.3155));

       (*расчет расхода газа*)
       //"Sensors".Q_gas.Value := "Sensors".Q_gas.a * "Sensors".Q_gas.Ksh * "Sensors".Q_gas.Kp * "Sensors".Q_gas.E * 3.1415926 * SQR("Sensors".Q_gas.d) / 4 * SQRT((2 * "Sensors".dP_gas_boiler.Value *1000* "Sensors".Q_gas.ros * "Sensors".Q_gas.Pgas *293.15) / ("Sensors".Q_gas.Ps * ("Sensors".Q_gas.Tgas + 273.15) * "Sensors".Q_gas.K)) * 3600 / "Sensors".Q_gas.ros;
       //"Sensors".Q_gas.Value := "Sensors".Q_gas.a * "Sensors".Q_gas.Ksh * "Sensors".Q_gas.Kp * "Sensors".Q_gas.E * 3.1415926 * SQR("Sensors".Q_gas.d) / 4 * SQRT((2 * "Sensors".dP_gas_boiler.Value * 1000 * "Sensors".Q_gas.ros * "Sensors".Q_gas.Pgas * 293.15) / ("Sensors".Q_gas.Ps * ("Sensors".Q_gas.Tgas + 273.15) * "Sensors".Q_gas.K)) * 3600 / "Sensors".Q_gas.ros;

       "Sensors".Q_gas.Value := ("Sensors".Q_gas."a" * "Sensors".Q_gas.Ksh * "Sensors".Q_gas.Kp * "Sensors".Q_gas."E" * 3.1415926 * (("Sensors".Q_gas.d) ** 2) / 4 * SQRT(2 * "Sensors".dP_gas_boiler.Value * 1000 * ("Sensors".Q_gas.ros * "Sensors".Q_gas.Pgas * 1000 * 293.15 / ("Sensors".Q_gas.Ps * ("Sensors".Q_gas.Tgas + 273.15) * "Sensors".Q_gas.K)))) * 3600 / "Sensors".Q_gas.ros;
       IF "Sensors".Q_gas.Value < 60.0 THEN
           "Sensors".Q_gas.Value := 0.0;
       END_IF;
   ELSE
       "Sensors".Q_gas.Value := 0;
   END_IF;


   //"Sensors".Q_gas.Value := (0.25 * "Sensors".Q_gas.a * "Sensors".Q_gas.Kp * (1 - ((0.351 + 0.256 * (("Sensors".Q_gas.d / "Sensors".Q_gas.Dtrub) ** 4)) + (0.93 * (("Sensors".Q_gas.d / "Sensors".Q_gas.Dtrub) ** 8))) * (1 - (1 - "Sensors".dP_gas_boiler.Value / 141.3232) ** (1 / 1.3155))) * 3.14159 * (("Sensors".Q_gas.d) ** 2) * SQRT(2 * "Sensors".dP_gas_boiler.Value * 1000 * ("Sensors".Q_gas.ros * 141.3232 * 1000 * 293.15 / (101.325 * 1000 * (-5 + 273.15) * 0.99832)))) / 0.67245 * 3600;
END_FUNCTION

FUNCTION "Read_sensor_4_20" : Void   // FC2, SCL
{ S7_Optimized_Access := 'TRUE' }
VERSION : 0.1
   VAR_INPUT
      Low_limit_phisical_current : Real;   // Нижний предел датчика в физической величине текущий
      High_limit_phisical_current : Real;   // Верхний предел датчика в физической величине текущий
      Low_limit_ADC_current : Int;   // Нижний предел датчика в АЦП текущий
      High_limit_ADC_current : Int;   // Верхний предел датчика в АЦП текущий
   END_VAR
   VAR_OUTPUT
      Current_ADC : Int;   // Текущий код АЦП
      Value : Real;   // Текущее значение в физической величине
      Alarm_sensor : Bool;   // Неисправность датчика
      Current : Real;   // Текущее значение тока
   END_VAR
   VAR_IN_OUT
      N_module : USInt;   // № модуля (начиная с 1)
      N_chanel : USInt;   // № канала (начиная с 1)
   END_VAR
   VAR_TEMP
      ADC : Int;   // Текущий код АЦП (для использования внутри функции)
      K : Real;   // Коэффициент К
      "B" : Real;   // Коэффициент B
   END_VAR
BEGIN
   (*проверка правильности введеного значения № Модуля*)
   IF #N_module < 1 OR #N_module > 3 THEN
       #N_module := 0;
   END_IF;

   (*проверка правильности введеного значения № Канала*)
   IF #N_module = 0 THEN
       #N_chanel := 0;
   ELSE
       IF #N_chanel < 1 OR #N_chanel > 8 THEN
           #N_chanel := 0;
       END_IF;
   END_IF;

   (*считывание кода АЦП выбранного канала*)
   CASE #N_module OF
       1:  // Модуль 1
           CASE #N_chanel OF
               1:  #ADC := "Module1Chanel1";   //Канал 1
               2:  #ADC := "Module1Chanel2";   //Канал 2
               3:  #ADC := "Module1Chanel3";   //Канал 3
               4:  #ADC := "Module1Chanel4";   //Канал 4
               5:  #ADC := "Module1Chanel5";   //Канал 5
               6:  #ADC := "Module1Chanel6";   //Канал 6
               7:  #ADC := "Module1Chanel7";   //Канал 7
               8:  #ADC := "Module1Chanel8";   //Канал 8
           ELSE
               #ADC := 0;
           END_CASE;
       2:  // Модуль 2
           CASE #N_chanel OF
               1:  #ADC := "Module2Chanel1";   //Канал 1
               2:  #ADC := "Module2Chanel2";   //Канал 2
               3:  #ADC := "Module2Chanel3";   //Канал 3
               4:  #ADC := "Module2Chanel4";   //Канал 4
               5:  #ADC := "Module2Chanel5";   //Канал 5
               6:  #ADC := "Module2Chanel6";   //Канал 6
               7:  #ADC := "Module2Chanel7";   //Канал 7
               8:  #ADC := "Module2Chanel8";   //Канал 8
           ELSE
               #ADC := 0;
       END_CASE;
       3:  // Модуль 3
           CASE #N_chanel OF
               1:  #ADC := "Module3Chanel1";   //Канал 1
               2:  #ADC := "Module3Chanel2";   //Канал 2
               3:  #ADC := "Module3Chanel3";   //Канал 3
               4:  #ADC := "Module3Chanel4";   //Канал 4
               5:  #ADC := "Module3Chanel5";   //Канал 5
               6:  #ADC := "Module3Chanel6";   //Канал 6
               7:  #ADC := "Module3Chanel7";   //Канал 7
               8:  #ADC := "Module3Chanel8";   //Канал 8
           ELSE
               #ADC := 0;
           END_CASE;
   ELSE
       #ADC := 0;
   END_CASE;
   #Current_ADC := #ADC;

   (*вычисление физического значения*)
   #K := (#High_limit_phisical_current - #Low_limit_phisical_current) / (#High_limit_ADC_current - #Low_limit_ADC_current);
   #"B" := #Low_limit_phisical_current - (#K * #Low_limit_ADC_current);
   IF #ADC < -4864 THEN
       #Value := -99999;
       #Alarm_sensor := true;
   END_IF;
   IF #ADC > 32511 THEN
       #Value := 99999;
       #Alarm_sensor := true;
   END_IF;
   IF #ADC >= -4864 AND #ADC <= 32511 THEN
       #Value := (#K * #ADC) + #"B";
       #Alarm_sensor := false;
   END_IF;

   (* (*проверка исправности датчика*)
   IF #ADC=32767 OR #ADC=-32768 THEN
       #Alarm_sensor := true;
   ELSE
       #Alarm_sensor := false;
   END_IF; *)

   (*вычисление физического значения тока*)
   #Current := (((20-4)/(INT_TO_REAL(27648 - 0)))*(INT_TO_REAL(#ADC)))+4;
END_FUNCTION

FUNCTION "Read_discret_signal" : Void   // FC3, SCL
{ S7_Optimized_Access := 'TRUE' }
VERSION : 0.1
   VAR_INPUT
      Invert : Bool;   // Необходимость инвертирования сигнала
   END_VAR
   VAR_OUTPUT
      Value : Bool;   // Текущее значение в физической величине
   END_VAR
   VAR_IN_OUT
      N_module : USInt;   // № модуля (начиная с 1)
      N_chanel : USInt;   // № канала (начиная с 1)
   END_VAR
   VAR_TEMP
      Signal : Bool;   // Текущее значение дискретного сигнала (для использования внутри функции)
   END_VAR
BEGIN
   (*проверка правильности введеного значения № Модуля*)
   IF #N_module < 4 OR #N_module > 9 THEN
       #N_module := 0;
   END_IF;

   (*проверка правильности введеного значения № Канала*)
   IF #N_module = 0 THEN
       #N_chanel := 0;
   ELSE
       IF #N_chanel < 1 OR #N_chanel > 16 THEN
           #N_chanel := 0;
       END_IF;
   END_IF;

